gfCNCPoint6[2430] = {X 578.0214, Y 47.7529, Z -8.0000, A 0.000, B 0.000, C 0.000 }
gfCNCPoint6[2431] = {X 577.4979, Y 46.9263, Z -8.0000, A 0.000, B 0.000, C 0.000 }
gfCNCPoint6[2432] = {X 577.4375, Y 46.7968, Z -8.0000, A 0.000, B 0.000, C 0.000 }
gfCNCPoint6[2433] = {X 577.3813, Y 46.6655, Z -8.0000, A 0.000, B 0.000, C 0.000 }
gfCNCPoint6[2434] = {X 572.1002, Y 33.7518, Z -8.0000, A 0.000, B 0.000, C 0.000 }
gfCNCPoint6[2435] = {X 572.1003, Y 35.0200, Z -8.0000, A 0.000, B 0.000, C 0.000 }
gfCNCPoint6[2436] = {X 572.1004, Y 40.7342, Z -8.0000, A 0.000, B 0.000, C 0.000 }
gfCNCPoint6[2437] = {X 572.7444, Y 41.4232, Z -8.0000, A 0.000, B 0.000, C 0.000 }
gfCNCPoint6[2438] = {X 573.2268, Y 42.2337, Z -8.0000, A 0.000, B 0.000, C 0.000 }
gfCNCPoint6[2439] = {X 573.5254, Y 43.1283, Z -8.0000, A 0.000, B 0.000, C 0.000 }
gfCNCPoint6[2440] = {X 573.6264, Y 44.0660, Z -8.0000, A 0.000, B 0.000, C 0.000 }
gfCNCPoint6[2441] = {X 573.6264, Y 45.0000, Z -8.0000, A 0.000, B 0.000, C 0.000 }
gfCNCPoint6[2442] = {X 573.5140, Y 45.9884, Z -8.0000, A 0.000, B 0.000, C 0.000 }
gfCNCPoint6[2443] = {X 573.1824, Y 46.9263, Z -8.0000, A 0.000, B 0.000, C 0.000 }
gfCNCPoint6[2444] = {X 572.6569, Y 47.7553, Z -8.0000, A 0.000, B 0.000, C 0.000 }
gfCNCPoint6[2445] = {X 571.9608, Y 48.4472, Z -8.0000, A 0.000, B 0.000, C 0.000 }
gfCNCPoint6[2446] = {X 571.1286, Y 48.9676, Z -8.0000, A 0.000, B 0.000, C 0.000 }
gfCNCPoint6[2447] = {X 570.2018, Y 49.2905, Z -8.0000, A 0.000, B 0.000, C 0.000 }
gfCNCPoint6[2448] = {X 569.2264, Y 49.4000, Z -8.0000, A 0.000, B 0.000, C 0.000 }
gfCNCPoint6[2449] = {X 562.4443, Y 49.4000, Z -8.0000, A 0.000, B 0.000, C 0.000 }
gfCNCPoint6[2450] = {X 561.4652, Y 49.2897, Z -8.0000, A 0.000, B 0.000, C 0.000 }
gfCNCPoint6[2451] = {X 560.5352, Y 48.9643, Z -8.0000, A 0.000, B 0.000, C 0.000 }
gfCNCPoint6[2452] = {X 559.7009, Y 48.4401, Z -8.0000, A 0.000, B 0.000, C 0.000 }
gfCNCPoint6[2453] = {X 559.0042, Y 47.7434, Z -8.0000, A 0.000, B 0.000, C 0.000 }
gfCNCPoint6[2454] = {X 558.4800, Y 46.9091, Z -8.0000, A 0.000, B 0.000, C 0.000 }
gfCNCPoint6[2455] = {X 558.1546, Y 45.9791, Z -8.0000, A 0.000, B 0.000, C 0.000 }
gfCNCPoint6[2456] = {X 558.0443, Y 45.0000, Z -8.0000, A 0.000, B 0.000, C 0.000 }
gfCNCPoint6[2457] = {X 558.0443, Y 44.0647, Z -8.0000, A 0.000, B 0.000, C 0.000 }
gfCNCPoint6[2458] = {X 558.1476, Y 43.1278, Z -8.0000, A 0.000, B 0.000, C 0.000 }
gfCNCPoint6[2459] = {X 558.4468, Y 42.2339, Z -8.0000, A 0.000, B 0.000, C 0.000 }
gfCNCPoint6[2460] = {X 558.9284, Y 41.4236, Z -8.0000, A 0.000, B 0.000, C 0.000 }
gfCNCPoint6[2461] = {X 559.5706, Y 40.7336, Z -8.0000, A 0.000, B 0.000, C 0.000 }
gfCNCPoint6[2462] = {X 559.5710, Y 9.2664, Z -8.0000, A 0.000, B 0.000, C 0.000 }
gfCNCPoint6[2463] = {X 558.9267, Y 8.5773, Z -8.0000, A 0.000, B 0.000, C 0.000 }
gfCNCPoint6[2464] = {X 558.4441, Y 7.7667, Z -8.0000, A 0.000, B 0.000, C 0.000 }
gfCNCPoint6[2465] = {X 558.1454, Y 6.8719, Z -8.0000, A 0.000, B 0.000, C 0.000 }
gfCNCPoint6[2466] = {X 558.0443, Y 5.9340, Z -8.0000, A 0.000, B 0.000, C 0.000 }
gfCNCPoint6[2467] = {X 558.0443, Y 5.0000, Z -8.0000, A 0.000, B 0.000, C 0.000 }
gfCNCPoint6[2468] = {X 558.1353, Y 4.1096, Z -8.0000, A 0.000, B 0.000, C 0.000 }
gfCNCPoint6[2469] = {X 558.4047, Y 3.2561, Z -8.0000, A 0.000, B 0.000, C 0.000 }
gfCNCPoint6[2470] = {X 558.9156, Y 2.3717, Z -8.0000, A 0.000, B 0.000, C 0.000 }
gfCNCPoint6[2471] = {X 559.6166, Y 1.6289, Z -8.0000, A 0.000, B 0.000, C 0.000 }
gfCNCPoint6[2472] = {X 560.4700, Y 1.0678, Z -8.0000, A 0.000, B 0.000, C 0.000 }
gfCNCPoint6[2473] = {X 561.4298, Y 0.7185, Z -8.0000, A 0.000, B 0.000, C 0.000 }
gfCNCPoint6[2474] = {X 562.4443, Y 0.6000, Z -8.0000, A 0.000, B 0.000, C 0.000 }
gfCNCPoint6[2475] = {X 570.9376, Y 0.6000, Z -8.0000, A 0.000, B 0.000, C 0.000 }
gfCNCPoint6[2476] = {X 571.9520, Y 0.7185, Z -8.0000, A 0.000, B 0.000, C 0.000 }
gfCNCPoint6[2477] = {X 572.9118, Y 1.0678, Z -8.0000, A 0.000, B 0.000, C 0.000 }
gfCNCPoint6[2478] = {X 573.7652, Y 1.6289, Z -8.0000, A 0.000, B 0.000, C 0.000 }
gfCNCPoint6[2479] = {X 574.4663, Y 2.3717, Z -8.0000, A 0.000, B 0.000, C 0.000 }
gfCNCPoint6[2480] = {X 574.9772, Y 3.2561, Z -8.0000, A 0.000, B 0.000, C 0.000 }
gfCNCPoint6[2481] = {X 575.2465, Y 4.1096, Z -8.0000, A 0.000, B 0.000, C 0.000 }
gfCNCPoint6[2482] = {X 575.3376, Y 5.0000, Z -8.0000, A 0.000, B 0.000, C 0.000 }
gfCNCPoint6[2483] = {X 575.3372, Y 5.9910, Z -8.0000, A 0.000, B 0.000, C 0.000 }
gfCNCPoint6[2484] = {X 575.2578, Y 6.7682, Z -8.0000, A 0.000, B 0.000, C 0.000 }
gfCNCPoint6[2485] = {X 575.0421, Y 7.5192, Z -8.0000, A 0.000, B 0.000, C 0.000 }
gfCNCPoint6[2486] = {X 574.6971, Y 8.2201, Z -8.0000, A 0.000, B 0.000, C 0.000 }
gfCNCPoint6[2487] = {X 575.2866, Y 9.6556, Z -8.0000, A 0.000, B 0.000, C 0.000 }
gfCNCPoint6[2488] = {X 578.9730, Y 18.7089, Z -8.0000, A 0.000, B 0.000, C 0.000 }
gfCNCPoint6[2489] = {X 580.9325, Y 23.5210, Z -8.0000, A 0.000, B 0.000, C 0.000 }
gfCNCPoint6[2490] = {X 581.1912, Y 24.1565, Z -8.0000, A 0.000, B 0.000, C 0.000 }
gfCNCPoint6[2491] = {X 581.4509, Y 23.5214, Z -8.0000, A 0.000, B 0.000, C 0.000 }
gfCNCPoint6[2492] = {X 587.7566, Y 8.0994, Z -8.0000, A 0.000, B 0.000, C 0.000 }
gfCNCPoint6[2493] = {X 587.4433, Y 7.4139, Z -8.0000, A 0.000, B 0.000, C 0.000 }
gfCNCPoint6[2494] = {X 587.2515, Y 6.6850, Z -8.0000, A 0.000, B 0.000, C 0.000 }
gfCNCPoint6[2495] = {X 587.1870, Y 5.9340, Z -8.0000, A 0.000, B 0.000, C 0.000 }
gfCNCPoint6[2496] = {X 587.1870, Y 5.0000, Z -8.0000, A 0.000, B 0.000, C 0.000 }
gfCNCPoint6[2497] = {X 587.2780, Y 4.1096, Z -8.0000, A 0.000, B 0.000, C 0.000 }
gfCNCPoint6[2498] = {X 587.5473, Y 3.2561, Z -8.0000, A 0.000, B 0.000, C 0.000 }
gfCNCPoint6[2499] = {X 588.0582, Y 2.3717, Z -8.0000, A 0.000, B 0.000, C 0.000 }
gfCNCPoint6[2500] = {X 588.7593, Y 1.6289, Z -8.0000, A 0.000, B 0.000, C 0.000 }
gfCNCPoint6[2501] = {X 589.6127, Y 1.0678, Z -8.0000, A 0.000, B 0.000, C 0.000 }
gfCNCPoint6[2502] = {X 590.5725, Y 0.7185, Z -8.0000, A 0.000, B 0.000, C 0.000 }
gfCNCPoint6[2503] = {X 591.5870, Y 0.6000, Z -8.0000, A 0.000, B 0.000, C 0.000 }
gfCNCPoint6[2504] = {X 600.0000, Y 0.6000, Z -8.0000, A 0.000, B 0.000, C 0.000 }
gfCNCPoint6[2505] = {X 600.8721, Y 0.6873, Z -8.0000, A 0.000, B 0.000, C 0.000 }
gfCNCPoint6[2506] = {X 601.7095, Y 0.9457, Z -8.0000, A 0.000, B 0.000, C 0.000 }
gfCNCPoint6[2507] = {X 602.4791, Y 1.3649, Z -8.0000, A 0.000, B 0.000, C 0.000 }
gfCNCPoint6[2508] = {X 603.1504, Y 1.9284, Z -8.0000, A 0.000, B 0.000, C 0.000 }
gfCNCPoint6[2509] = {X 603.6967, Y 2.6137, Z -8.0000, A 0.000, B 0.000, C 0.000 }
gfCNCPoint6[2510] = {X 603.6967, Y 1.8143, Z -8.0000, A 0.000, B 0.000, C 0.000 }
gfCNCPoint6[2511] = {X 602.9514, Y 1.1137, Z -8.0000, A 0.000, B 0.000, C 0.000 }
gfCNCPoint6[2512] = {X 602.0764, Y 0.5838, Z -8.0000, A 0.000, B 0.000, C 0.000 }
gfCNCPoint6[2513] = {X 601.1102, Y 0.2480, Z -8.0000, A 0.000, B 0.000, C 0.000 }
gfCNCPoint6[2514] = {X 600.0953, Y 0.1209, Z -8.0000, A 0.000, B 0.000, C 0.000 }
gfCNCPoint6[2515] = {X 600.0950, Y -0.0186, Z -8.0000, A 0.000, B 0.000, C 0.000 }
gfCNCPoint6[2516] = {X 600.0672, Y -0.0699, Z -8.0000, A 0.000, B 0.000, C 0.000 }
gfCNCPoint6[2517] = {X 600.0147, Y -0.0952, Z -8.0000, A 0.000, B 0.000, C 0.000 }
gfCNCPoint6[2518] = {X 580.1328, Y -0.0952, Z -8.0000, A 0.000, B 0.000, C 0.000 }
gfCNCPoint6[2519] = {X 580.1328, Y 4.7048, Z -8.0000, A 0.000, B 0.000, C 0.000 }
gfCNCPoint6[2520] = {X 580.1364, Y 4.8524, Z -8.0000, A 0.000, B 0.000, C 0.000 }
gfCNCPoint6[2521] = {X 580.1376, Y 5.0000, Z -8.0000, A 0.000, B 0.000, C 0.000 }
gfCNCPoint6[2522] = {X 580.1376, Y 5.9339, Z -8.0000, A 0.000, B 0.000, C 0.000 }
gfCNCPoint6[2523] = {X 580.0686, Y 7.0584, Z -8.0000, A 0.000, B 0.000, C 0.000 }
gfCNCPoint6[2524] = {X 579.8627, Y 8.1660, Z -8.0000, A 0.000, B 0.000, C 0.000 }
gfCNCPoint6[2525] = {X 581.2004, Y 11.4512, Z -8.0000, A 0.000, B 0.000, C 0.000 }
gfCNCPoint6[2526] = {X 582.6182, Y 7.9837, Z -8.0000, A 0.000, B 0.000, C 0.000 }
gfCNCPoint6[2527] = {X 582.4488, Y 6.9991, Z -8.0000, A 0.000, B 0.000, C 0.000 }
gfCNCPoint6[2528] = {X 582.3872, Y 6.0018, Z -8.0000, A 0.000, B 0.000, C 0.000 }
gfCNCPoint6[2529] = {X 582.3870, Y 5.0000, Z -8.0000, A 0.000, B 0.000, C 0.000 }
gfCNCPoint6[2530] = {X 582.3881, Y 4.8524, Z -8.0000, A 0.000, B 0.000, C 0.000 }
gfCNCPoint6[2531] = {X 582.3917, Y 4.7048, Z -8.0000, A 0.000, B 0.000, C 0.000 }
gfCNCPoint6[2532] = {X 580.1328, Y 4.7048, Z -8.0000, A 0.000, B 0.000, C 0.000 }
gfCNCPoint6[2533] = {X 580.1328, Y 2.3048, Z -8.0000, A 0.000, B 0.000, C 0.000 }
gfCNCPoint6[2534] = {X 577.1806, Y 2.3048, Z -8.0000, A 0.000, B 0.000, C 0.000 }
gfCNCPoint6[2535] = {X 577.5739, Y 3.5173, Z -8.0000, A 0.000, B 0.000, C 0.000 }
gfCNCPoint6[2536] = {X 577.7341, Y 4.7818, Z -8.0000, A 0.000, B 0.000, C 0.000 }
gfCNCPoint6[2537] = {X 577.7367, Y 4.8909, Z -8.0000, A 0.000, B 0.000, C 0.000 }
gfCNCPoint6[2538] = {X 577.7376, Y 5.0000, Z -8.0000, A 0.000, B 0.000, C 0.000 }
gfCNCPoint6[2539] = {X 577.7376, Y 5.9339, Z -8.0000, A 0.000, B 0.000, C 0.000 }
gfCNCPoint6[2540] = {X 577.6319, Y 7.1280, Z -8.0000, A 0.000, B 0.000, C 0.000 }
gfCNCPoint6[2541] = {X 577.3182, Y 8.2850, Z -8.0000, A 0.000, B 0.000, C 0.000 }
gfCNCPoint6[2542] = {X 577.5061, Y 8.7426, Z -8.0000, A 0.000, B 0.000, C 0.000 }
gfCNCPoint6[2543] = {X 581.1958, Y 17.8038, Z -8.0000, A 0.000, B 0.000, C 0.000 }
gfCNCPoint6[2544] = {X 585.1513, Y 8.1300, Z -8.0000, A 0.000, B 0.000, C 0.000 }
gfCNCPoint6[2545] = {X 584.8834, Y 7.0753, Z -8.0000, A 0.000, B 0.000, C 0.000 }
gfCNCPoint6[2546] = {X 584.7872, Y 5.9914, Z -8.0000, A 0.000, B 0.000, C 0.000 }
gfCNCPoint6[2547] = {X 584.7870, Y 5.0000, Z -8.0000, A 0.000, B 0.000, C 0.000 }
gfCNCPoint6[2548] = {X 584.7878, Y 4.8909, Z -8.0000, A 0.000, B 0.000, C 0.000 }
gfCNCPoint6[2549] = {X 584.7905, Y 4.7818, Z -8.0000, A 0.000, B 0.000, C 0.000 }
gfCNCPoint6[2550] = {X 584.9506, Y 3.5173, Z -8.0000, A 0.000, B 0.000, C 0.000 }
gfCNCPoint6[2551] = {X 585.3439, Y 2.3048, Z -8.0000, A 0.000, B 0.000, C 0.000 }
gfCNCPoint6[2552] = {X 580.1328, Y 2.3048, Z -8.0000, A 0.000, B 0.000, C 0.000 }
gfCNCPoint6[2553] = {X 580.1328, Y -0.0952, Z -8.0000, A 0.000, B 0.000, C 0.000 }
gfCNCPoint6[2554] = {X 351.5709, Y -0.0952, Z -8.0000, A 0.000, B 0.000, C 0.000 }
gfCNCPoint6[2555] = {X 351.4056, Y -0.1263, Z -8.0000, A 0.000, B 0.000, C 0.000 }
gfCNCPoint6[2556] = {X 348.9077, Y -0.4729, Z -8.0000, A 0.000, B 0.000, C 0.000 }
gfCNCPoint6[2557] = {X 346.3883, Y -0.5836, Z -8.0000, A 0.000, B 0.000, C 0.000 }
gfCNCPoint6[2558] = {X 343.8697, Y -0.4573, Z -8.0000, A 0.000, B 0.000, C 0.000 }
gfCNCPoint6[2559] = {X 341.3740, Y -0.0952, Z -8.0000, A 0.000, B 0.000, C 0.000 }
gfCNCPoint6[2560] = {X -0.0147, Y -0.0952, Z -8.0000, A 0.000, B 0.000, C 0.000 }
gfCNCPoint6[2561] = {X -0.0672, Y -0.0699, Z -8.0000, A 0.000, B 0.000, C 0.000 }
gfCNCPoint6[2562] = {X -0.0950, Y -0.0186, Z -8.0000, A 0.000, B 0.000, C 0.000 }
gfCNCPoint6[2563] = {X -0.0967, Y 0.8568, Z -8.0000, A 0.000, B 0.000, C 0.000 }
gfCNCPoint6[2564] = {X -0.0967, Y 8.7891, Z -8.0000, A 0.000, B 0.000, C 0.000 }
gfCNCPoint6[2565] = {X -0.7634, Y 8.9979, Z -8.0000, A 0.000, B 0.000, C 0.000 }
gfCNCPoint6[2566] = {X -1.3934, Y 9.2998, Z -8.0000, A 0.000, B 0.000, C 0.000 }
gfCNCPoint6[2567] = {X -1.9904, Y 9.6404, Z -8.0000, A 0.000, B 0.000, C 0.000 }
gfCNCPoint6[2568] = {X -2.6455, Y 10.0885, Z -8.0000, A 0.000, B 0.000, C 0.000 }
gfCNCPoint6[2569] = {X -3.2194, Y 10.6368, Z -8.0000, A 0.000, B 0.000, C 0.000 }
gfCNCPoint6[2570] = {X -3.6967, Y 11.2708, Z -8.0000, A 0.000, B 0.000, C 0.000 }
gfCNCPoint6[2571] = {X -3.6967, Y 12.3466, Z -8.0000, A 0.000, B 0.000, C 0.000 }
gfCNCPoint6[2572] = {X -3.2334, Y 11.4386, Z -8.0000, A 0.000, B 0.000, C 0.000 }
gfCNCPoint6[2573] = {X -2.5735, Y 10.6616, Z -8.0000, A 0.000, B 0.000, C 0.000 }
gfCNCPoint6[2574] = {X -1.7526, Y 10.0573, Z -8.0000, A 0.000, B 0.000, C 0.000 }
gfCNCPoint6[2575] = {X -1.0994, Y 9.6852, Z -8.0000, A 0.000, B 0.000, C 0.000 }
gfCNCPoint6[2576] = {X -0.1608, Y 9.3012, Z -8.0000, A 0.000, B 0.000, C 0.000 }
gfCNCPoint6[2577] = {X 0.8408, Y 9.1423, Z -8.0000, A 0.000, B 0.000, C 0.000 }
gfCNCPoint6[2578] = {X 1.8521, Y 9.2169, Z -8.0000, A 0.000, B 0.000, C 0.000 }
gfCNCPoint6[2579] = {X 2.2301, Y 9.3067, Z -8.0000, A 0.000, B 0.000, C 0.000 }
gfCNCPoint6[2580] = {X 2.5987, Y 9.4295, Z -8.0000, A 0.000, B 0.000, C 0.000 }
gfCNCPoint6[2581] = {X 3.4585, Y 9.0449, Z -8.0000, A 0.000, B 0.000, C 0.000 }
gfCNCPoint6[2582] = {X 5.5423, Y 8.2600, Z -8.0000, A 0.000, B 0.000, C 0.000 }
gfCNCPoint6[2583] = {X 7.6901, Y 7.6725, Z -8.0000, A 0.000, B 0.000, C 0.000 }
gfCNCPoint6[2584] = {X 9.8833, Y 7.2876, Z -8.0000, A 0.000, B 0.000, C 0.000 }
gfCNCPoint6[2585] = {X 12.1029, Y 7.1087, Z -8.0000, A 0.000, B 0.000, C 0.000 }
gfCNCPoint6[2586] = {X 14.3294, Y 7.1373, Z -8.0000, A 0.000, B 0.000, C 0.000 }
gfCNCPoint6[2587] = {X 16.5436, Y 7.3732, Z -8.0000, A 0.000, B 0.000, C 0.000 }
gfCNCPoint6[2588] = {X 18.2874, Y 7.7294, Z -8.0000, A 0.000, B 0.000, C 0.000 }
gfCNCPoint6[2589] = {X 19.9860, Y 8.2610, Z -8.0000, A 0.000, B 0.000, C 0.000 }
gfCNCPoint6[2590] = {X 21.6217, Y 8.9626, Z -8.0000, A 0.000, B 0.000, C 0.000 }
gfCNCPoint6[2591] = {X 23.1776, Y 9.8268, Z -8.0000, A 0.000, B 0.000, C 0.000 }
gfCNCPoint6[2592] = {X 24.6376, Y 10.8447, Z -8.0000, A 0.000, B 0.000, C 0.000 }
gfCNCPoint6[2593] = {X 25.7303, Y 11.8004, Z -8.0000, A 0.000, B 0.000, C 0.000 }
gfCNCPoint6[2594] = {X 26.7104, Y 12.8713, Z -8.0000, A 0.000, B 0.000, C 0.000 }
gfCNCPoint6[2595] = {X 27.5658, Y 14.0441, Z -8.0000, A 0.000, B 0.000, C 0.000 }
gfCNCPoint6[2596] = {X 28.2861, Y 15.3044, Z -8.0000, A 0.000, B 0.000, C 0.000 }
gfCNCPoint6[2597] = {X 28.8624, Y 16.6368, Z -8.0000, A 0.000, B 0.000, C 0.000 }
gfCNCPoint6[2598] = {X 29.3390, Y 18.3013, Z -8.0000, A 0.000, B 0.000, C 0.000 }
gfCNCPoint6[2599] = {X 29.6217, Y 20.0095, Z -8.0000, A 0.000, B 0.000, C 0.000 }
gfCNCPoint6[2600] = {X 29.7069, Y 21.7388, Z -8.0000, A 0.000, B 0.000, C 0.000 }
gfCNCPoint6[2601] = {X 29.5934, Y 23.4664, Z -8.0000, A 0.000, B 0.000, C 0.000 }
gfCNCPoint6[2602] = {X 29.2828, Y 25.1698, Z -8.0000, A 0.000, B 0.000, C 0.000 }
gfCNCPoint6[2603] = {X 28.7910, Y 26.7456, Z -8.0000, A 0.000, B 0.000, C 0.000 }
gfCNCPoint6[2604] = {X 28.0838, Y 28.2372, Z -8.0000, A 0.000, B 0.000, C 0.000 }
gfCNCPoint6[2605] = {X 27.1749, Y 29.6152, Z -8.0000, A 0.000, B 0.000, C 0.000 }
gfCNCPoint6[2606] = {X 26.3579, Y 30.5723, Z -8.0000, A 0.000, B 0.000, C 0.000 }
gfCNCPoint6[2607] = {X 25.4435, Y 31.4368, Z -8.0000, A 0.000, B 0.000, C 0.000 }
gfCNCPoint6[2608] = {X 25.6940, Y 31.5324, Z -8.0000, A 0.000, B 0.000, C 0.000 }
gfCNCPoint6[2609] = {X 25.9383, Y 31.6432, Z -8.0000, A 0.000, B 0.000, C 0.000 }
gfCNCPoint6[2610] = {X 26.6629, Y 32.0904, Z -8.0000, A 0.000, B 0.000, C 0.000 }
gfCNCPoint6[2611] = {X 27.2878, Y 32.6689, Z -8.0000, A 0.000, B 0.000, C 0.000 }
gfCNCPoint6[2612] = {X 27.6592, Y 33.1494, Z -8.0000, A 0.000, B 0.000, C 0.000 }
gfCNCPoint6[2613] = {X 27.9608, Y 33.6765, Z -8.0000, A 0.000, B 0.000, C 0.000 }
gfCNCPoint6[2614] = {X 30.9820, Y 39.9182, Z -8.0000, A 0.000, B 0.000, C 0.000 }
gfCNCPoint6[2615] = {X 31.3085, Y 40.8441, Z -8.0000, A 0.000, B 0.000, C 0.000 }
gfCNCPoint6[2616] = {X 31.4215, Y 41.8194, Z -8.0000, A 0.000, B 0.000, C 0.000 }
gfCNCPoint6[2617] = {X 31.3155, Y 42.7955, Z -8.0000, A 0.000, B 0.000, C 0.000 }
gfCNCPoint6[2618] = {X 30.9956, Y 43.7238, Z -8.0000, A 0.000, B 0.000, C 0.000 }
gfCNCPoint6[2619] = {X 30.4779, Y 44.5580, Z -8.0000, A 0.000, B 0.000, C 0.000 }
gfCNCPoint6[2620] = {X 29.7880, Y 45.2567, Z -8.0000, A 0.000, B 0.000, C 0.000 }
gfCNCPoint6[2621] = {X 29.2521, Y 45.6900, Z -8.0000, A 0.000, B 0.000, C 0.000 }
gfCNCPoint6[2622] = {X 28.5416, Y 46.1592, Z -8.0000, A 0.000, B 0.000, C 0.000 }
gfCNCPoint6[2623] = {X 27.7541, Y 46.4832, Z -8.0000, A 0.000, B 0.000, C 0.000 }
gfCNCPoint6[2624] = {X 26.9190, Y 46.6497, Z -8.0000, A 0.000, B 0.000, C 0.000 }
gfCNCPoint6[2625] = {X 26.0675, Y 46.6526, Z -8.0000, A 0.000, B 0.000, C 0.000 }
gfCNCPoint6[2626] = {X 25.2313, Y 46.4918, Z -8.0000, A 0.000, B 0.000, C 0.000 }
gfCNCPoint6[2627] = {X 23.4347, Y 47.4365, Z -8.0000, A 0.000, B 0.000, C 0.000 }
gfCNCPoint6[2628] = {X 21.5774, Y 48.2554, Z -8.0000, A 0.000, B 0.000, C 0.000 }
gfCNCPoint6[2629] = {X 19.6682, Y 48.9447, Z -8.0000, A 0.000, B 0.000, C 0.000 }
gfCNCPoint6[2630] = {X 17.7217, Y 49.4942, Z -8.0000, A 0.000, B 0.000, C 0.000 }
gfCNCPoint6[2631] = {X 15.7341, Y 49.8692, Z -8.0000, A 0.000, B 0.000, C 0.000 }
gfCNCPoint6[2632] = {X 13.7212, Y 50.0669, Z -8.0000, A 0.000, B 0.000, C 0.000 }
gfCNCPoint6[2633] = {X 11.6986, Y 50.0856, Z -8.0000, A 0.000, B 0.000, C 0.000 }
gfCNCPoint6[2634] = {X 9.6824, Y 49.9253, Z -8.0000, A 0.000, B 0.000, C 0.000 }
gfCNCPoint6[2635] = {X 7.6882, Y 49.5872, Z -8.0000, A 0.000, B 0.000, C 0.000 }
gfCNCPoint6[2636] = {X 6.2182, Y 49.2062, Z -8.0000, A 0.000, B 0.000, C 0.000 }
gfCNCPoint6[2637] = {X 4.7886, Y 48.6940, Z -8.0000, A 0.000, B 0.000, C 0.000 }
gfCNCPoint6[2638] = {X 3.4111, Y 48.0546, Z -8.0000, A 0.000, B 0.000, C 0.000 }
gfCNCPoint6[2639] = {X 1.9573, Y 47.2030, Z -8.0000, A 0.000, B 0.000, C 0.000 }
gfCNCPoint6[2640] = {X 0.5963, Y 46.2099, Z -8.0000, A 0.000, B 0.000, C 0.000 }
gfCNCPoint6[2641] = {X -0.5425, Y 45.1859, Z -8.0000, A 0.000, B 0.000, C 0.000 }
gfCNCPoint6[2642] = {X -1.5540, Y 44.0360, Z -8.0000, A 0.000, B 0.000, C 0.000 }
gfCNCPoint6[2643] = {X -2.4244, Y 42.7759, Z -8.0000, A 0.000, B 0.000, C 0.000 }
gfCNCPoint6[2644] = {X -3.1419, Y 41.4230, Z -8.0000, A 0.000, B 0.000, C 0.000 }
gfCNCPoint6[2645] = {X -3.6967, Y 39.9955, Z -8.0000, A 0.000, B 0.000, C 0.000 }
gfCNCPoint6[2646] = {X -3.6967, Y 41.3567, Z -8.0000, A 0.000, B 0.000, C 0.000 }
gfCNCPoint6[2647] = {X -3.0106, Y 42.7271, Z -8.0000, A 0.000, B 0.000, C 0.000 }
gfCNCPoint6[2648] = {X -2.1745, Y 44.0116, Z -8.0000, A 0.000, B 0.000, C 0.000 }
gfCNCPoint6[2649] = {X -1.1991, Y 45.1937, Z -8.0000, A 0.000, B 0.000, C 0.000 }
gfCNCPoint6[2650] = {X -0.0967, Y 46.2584, Z -8.0000, A 0.000, B 0.000, C 0.000 }
gfCNCPoint6[2651] = {X -0.0967, Y 99.1432, Z -8.0000, A 0.000, B 0.000, C 0.000 }
gfCNCPoint6[2652] = {X -0.0950, Y 100.0186, Z -8.0000, A 0.000, B 0.000, C 0.000 }
gfCNCPoint6[2653] = {X -0.0672, Y 100.0699, Z -8.0000, A 0.000, B 0.000, C 0.000 }
gfCNCPoint6[2654] = {X -0.0147, Y 100.0952, Z -8.0000, A 0.000, B 0.000, C 0.000 }
gfCNCPoint6[2655] = {X 120.5927, Y 100.0952, Z -8.0000, A 0.000, B 0.000, C 0.000 }
gfCNCPoint6[2656] = {X 121.0614, Y 100.8813, Z -8.0000, A 0.000, B 0.000, C 0.000 }
gfCNCPoint6[2657] = {X 121.6688, Y 101.5661, Z -8.0000, A 0.000, B 0.000, C 0.000 }
gfCNCPoint6[2658] = {X 122.3933, Y 102.1255, Z -8.0000, A 0.000, B 0.000, C 0.000 }
gfCNCPoint6[2659] = {X 123.2095, Y 102.5397, Z -8.0000, A 0.000, B 0.000, C 0.000 }
gfCNCPoint6[2660] = {X 124.0887, Y 102.7942, Z -8.0000, A 0.000, B 0.000, C 0.000 }
gfCNCPoint6[2661] = {X 125.0000, Y 102.8800, Z -8.0000, A 0.000, B 0.000, C 0.000 }
gfCNCPoint6[2662] = {X 143.7791, Y 102.8800, Z -8.0000, A 0.000, B 0.000, C 0.000 }
gfCNCPoint6[2663] = {X 144.6904, Y 102.7942, Z -8.0000, A 0.000, B 0.000, C 0.000 }
gfCNCPoint6[2664] = {X 145.5696, Y 102.5397, Z -8.0000, A 0.000, B 0.000, C 0.000 }
gfCNCPoint6[2665] = {X 146.3858, Y 102.1255, Z -8.0000, A 0.000, B 0.000, C 0.000 }
gfCNCPoint6[2666] = {X 147.1104, Y 101.5661, Z -8.0000, A 0.000, B 0.000, C 0.000 }
gfCNCPoint6[2667] = {X 147.7177, Y 100.8813, Z -8.0000, A 0.000, B 0.000, C 0.000 }
gfCNCPoint6[2668] = {X 148.1865, Y 100.0952, Z -8.0000, A 0.000, B 0.000, C 0.000 }
gfCNCPoint6[2669] = {X 150.8390, Y 100.0952, Z -8.0000, A 0.000, B 0.000, C 0.000 }
gfCNCPoint6[2670] = {X 150.8390, Y 95.2952, Z -8.0000, A 0.000, B 0.000, C 0.000 }
gfCNCPoint6[2671] = {X 187.9256, Y 95.2952, Z -8.0000, A 0.000, B 0.000, C 0.000 }
gfCNCPoint6[2672] = {X 187.9777, Y 95.0991, Z -8.0000, A 0.000, B 0.000, C 0.000 }
gfCNCPoint6[2673] = {X 188.0352, Y 94.9045, Z -8.0000, A 0.000, B 0.000, C 0.000 }
gfCNCPoint6[2674] = {X 187.2619, Y 94.0602, Z -8.0000, A 0.000, B 0.000, C 0.000 }
gfCNCPoint6[2675] = {X 151.4055, Y 94.0602, Z -8.0000, A 0.000, B 0.000, C 0.000 }
gfCNCPoint6[2676] = {X 150.7069, Y 94.8343, Z -8.0000, A 0.000, B 0.000, C 0.000 }
gfCNCPoint6[2677] = {X 150.7767, Y 95.0636, Z -8.0000, A 0.000, B 0.000, C 0.000 }
gfCNCPoint6[2678] = {X 150.8390, Y 95.2952, Z -8.0000, A 0.000, B 0.000, C 0.000 }
gfCNCPoint6[2679] = {X 150.8390, Y 97.6952, Z -8.0000, A 0.000, B 0.000, C 0.000 }
gfCNCPoint6[2680] = {X 190.1070, Y 97.6952, Z -8.0000, A 0.000, B 0.000, C 0.000 }
gfCNCPoint6[2681] = {X 190.1070, Y 97.0659, Z -8.0000, A 0.000, B 0.000, C 0.000 }
gfCNCPoint6[2682] = {X 190.1938, Y 96.1495, Z -8.0000, A 0.000, B 0.000, C 0.000 }
gfCNCPoint6[2683] = {X 190.4511, Y 95.2657, Z -8.0000, A 0.000, B 0.000, C 0.000 }
gfCNCPoint6[2684] = {X 190.8699, Y 94.4460, Z -8.0000, A 0.000, B 0.000, C 0.000 }
gfCNCPoint6[2685] = {X 188.3182, Y 91.6602, Z -8.0000, A 0.000, B 0.000, C 0.000 }
gfCNCPoint6[2686] = {X 150.3387, Y 91.6602, Z -8.0000, A 0.000, B 0.000, C 0.000 }
gfCNCPoint6[2687] = {X 147.8648, Y 94.4010, Z -8.0000, A 0.000, B 0.000, C 0.000 }
gfCNCPoint6[2688] = {X 148.2994, Y 95.2322, Z -8.0000, A 0.000, B 0.000, C 0.000 }
gfCNCPoint6[2689] = {X 148.5675, Y 96.1310, Z -8.0000, A 0.000, B 0.000, C 0.000 }
gfCNCPoint6[2690] = {X 148.6591, Y 97.0644, Z -8.0000, A 0.000, B 0.000, C 0.000 }
gfCNCPoint6[2691] = {X 148.6591, Y 97.6952, Z -8.0000, A 0.000, B 0.000, C 0.000 }
gfCNCPoint6[2692] = {X 150.8390, Y 97.6952, Z -8.0000, A 0.000, B 0.000, C 0.000 }
gfCNCPoint6[2693] = {X 150.8390, Y 100.0952, Z -8.0000, A 0.000, B 0.000, C 0.000 }
gfCNCPoint6[2694] = {X 190.5796, Y 100.0952, Z -8.0000, A 0.000, B 0.000, C 0.000 }
gfCNCPoint6[2695] = {X 191.0484, Y 100.8813, Z -8.0000, A 0.000, B 0.000, C 0.000 }
gfCNCPoint6[2696] = {X 191.6557, Y 101.5661, Z -8.0000, A 0.000, B 0.000, C 0.000 }
gfCNCPoint6[2697] = {X 192.3802, Y 102.1255, Z -8.0000, A 0.000, B 0.000, C 0.000 }
gfCNCPoint6[2698] = {X 193.1965, Y 102.5397, Z -8.0000, A 0.000, B 0.000, C 0.000 }
gfCNCPoint6[2699] = {X 194.0757, Y 102.7942, Z -8.0000, A 0.000, B 0.000, C 0.000 }
gfCNCPoint6[2700] = {X 194.9870, Y 102.8800, Z -8.0000, A 0.000, B 0.000, C 0.000 }
gfCNCPoint6[2701] = {X 212.6141, Y 102.8800, Z -8.0000, A 0.000, B 0.000, C 0.000 }
gfCNCPoint6[2702] = {X 213.0066, Y 102.8642, Z -8.0000, A 0.000, B 0.000, C 0.000 }
gfCNCPoint6[2703] = {X 213.3966, Y 102.8169, Z -8.0000, A 0.000, B 0.000, C 0.000 }
gfCNCPoint6[2704] = {X 213.7865, Y 102.8642, Z -8.0000, A 0.000, B 0.000, C 0.000 }
gfCNCPoint6[2705] = {X 214.1790, Y 102.8800, Z -8.0000, A 0.000, B 0.000, C 0.000 }
gfCNCPoint6[2706] = {X 233.4798, Y 102.8800, Z -8.0000, A 0.000, B 0.000, C 0.000 }
gfCNCPoint6[2707] = {X 234.3911, Y 102.7942, Z -8.0000, A 0.000, B 0.000, C 0.000 }
gfCNCPoint6[2708] = {X 235.2703, Y 102.5397, Z -8.0000, A 0.000, B 0.000, C 0.000 }
gfCNCPoint6[2709] = {X 236.0865, Y 102.1255, Z -8.0000, A 0.000, B 0.000, C 0.000 }
gfCNCPoint6[2710] = {X 236.8110, Y 101.5661, Z -8.0000, A 0.000, B 0.000, C 0.000 }
gfCNCPoint6[2711] = {X 237.4184, Y 100.8813, Z -8.0000, A 0.000, B 0.000, C 0.000 }
gfCNCPoint6[2712] = {X 237.8871, Y 100.0952, Z -8.0000, A 0.000, B 0.000, C 0.000 }
gfCNCPoint6[2713] = {X 261.4882, Y 100.0952, Z -8.0000, A 0.000, B 0.000, C 0.000 }
gfCNCPoint6[2714] = {X 261.4882, Y 90.4952, Z -8.0000, A 0.000, B 0.000, C 0.000 }
gfCNCPoint6[2715] = {X 266.0961, Y 90.4952, Z -8.0000, A 0.000, B 0.000, C 0.000 }
gfCNCPoint6[2716] = {X 266.1751, Y 90.3748, Z -8.0000, A 0.000, B 0.000, C 0.000 }
gfCNCPoint6[2717] = {X 266.2556, Y 90.2554, Z -8.0000, A 0.000, B 0.000, C 0.000 }
gfCNCPoint6[2718] = {X 263.5169, Y 89.1818, Z -8.0000, A 0.000, B 0.000, C 0.000 }
gfCNCPoint6[2719] = {X 261.4882, Y 90.4952, Z -8.0000, A 0.000, B 0.000, C 0.000 }
gfCNCPoint6[2720] = {X 261.4882, Y 92.8952, Z -8.0000, A 0.000, B 0.000, C 0.000 }
gfCNCPoint6[2721] = {X 267.4973, Y 92.8952, Z -8.0000, A 0.000, B 0.000, C 0.000 }
gfCNCPoint6[2722] = {X 267.8429, Y 92.2376, Z -8.0000, A 0.000, B 0.000, C 0.000 }
gfCNCPoint6[2723] = {X 268.2378, Y 91.6085, Z -8.0000, A 0.000, B 0.000, C 0.000 }
gfCNCPoint6[2724] = {X 269.1700, Y 90.4463, Z -8.0000, A 0.000, B 0.000, C 0.000 }
gfCNCPoint6[2725] = {X 270.2694, Y 89.4409, Z -8.0000, A 0.000, B 0.000, C 0.000 }
gfCNCPoint6[2726] = {X 270.2694, Y 89.2510, Z -8.0000, A 0.000, B 0.000, C 0.000 }
gfCNCPoint6[2727] = {X 263.2463, Y 86.4979, Z -8.0000, A 0.000, B 0.000, C 0.000 }
gfCNCPoint6[2728] = {X 253.3650, Y 92.8952, Z -8.0000, A 0.000, B 0.000, C 0.000 }
gfCNCPoint6[2729] = {X 261.4882, Y 92.8952, Z -8.0000, A 0.000, B 0.000, C 0.000 }
gfCNCPoint6[2730] = {X 261.4882, Y 95.2952, Z -8.0000, A 0.000, B 0.000, C 0.000 }
gfCNCPoint6[2731] = {X 269.1713, Y 95.2952, Z -8.0000, A 0.000, B 0.000, C 0.000 }
gfCNCPoint6[2732] = {X 269.5515, Y 94.1746, Z -8.0000, A 0.000, B 0.000, C 0.000 }
gfCNCPoint6[2733] = {X 270.1082, Y 93.1304, Z -8.0000, A 0.000, B 0.000, C 0.000 }
gfCNCPoint6[2734] = {X 270.8267, Y 92.1902, Z -8.0000, A 0.000, B 0.000, C 0.000 }
gfCNCPoint6[2735] = {X 271.6880, Y 91.3788, Z -8.0000, A 0.000, B 0.000, C 0.000 }
gfCNCPoint6[2736] = {X 272.6694, Y 90.7176, Z -8.0000, A 0.000, B 0.000, C 0.000 }
gfCNCPoint6[2737] = {X 272.6694, Y 87.6139, Z -8.0000, A 0.000, B 0.000, C 0.000 }
gfCNCPoint6[2738] = {X 262.9757, Y 83.8140, Z -8.0000, A 0.000, B 0.000, C 0.000 }
gfCNCPoint6[2739] = {X 245.2418, Y 95.2952, Z -8.0000, A 0.000, B 0.000, C 0.000 }
gfCNCPoint6[2740] = {X 261.4882, Y 95.2952, Z -8.0000, A 0.000, B 0.000, C 0.000 }
gfCNCPoint6[2741] = {X 261.4882, Y 97.6952, Z -8.0000, A 0.000, B 0.000, C 0.000 }
gfCNCPoint6[2742] = {X 271.3527, Y 97.6952, Z -8.0000, A 0.000, B 0.000, C 0.000 }
gfCNCPoint6[2743] = {X 271.3529, Y 97.0186, Z -8.0000, A 0.000, B 0.000, C 0.000 }
gfCNCPoint6[2744] = {X 271.4810, Y 95.9545, Z -8.0000, A 0.000, B 0.000, C 0.000 }
gfCNCPoint6[2745] = {X 271.8382, Y 94.9440, Z -8.0000, A 0.000, B 0.000, C 0.000 }
gfCNCPoint6[2746] = {X 272.4074, Y 94.0359, Z -8.0000, A 0.000, B 0.000, C 0.000 }
gfCNCPoint6[2747] = {X 273.1610, Y 93.2739, Z -8.0000, A 0.000, B 0.000, C 0.000 }
gfCNCPoint6[2748] = {X 274.0629, Y 92.6949, Z -8.0000, A 0.000, B 0.000, C 0.000 }
gfCNCPoint6[2749] = {X 275.0694, Y 92.3266, Z -8.0000, A 0.000, B 0.000, C 0.000 }
gfCNCPoint6[2750] = {X 275.0694, Y 85.9769, Z -8.0000, A 0.000, B 0.000, C 0.000 }
gfCNCPoint6[2751] = {X 262.7051, Y 81.1301, Z -8.0000, A 0.000, B 0.000, C 0.000 }
gfCNCPoint6[2752] = {X 238.3590, Y 96.8921, Z -8.0000, A 0.000, B 0.000, C 0.000 }
gfCNCPoint6[2753] = {X 238.3598, Y 97.6952, Z -8.0000, A 0.000, B 0.000, C 0.000 }
gfCNCPoint6[2754] = {X 261.4882, Y 97.6952, Z -8.0000, A 0.000, B 0.000, C 0.000 }
gfCNCPoint6[2755] = {X 261.4882, Y 100.0952, Z -8.0000, A 0.000, B 0.000, C 0.000 }
gfCNCPoint6[2756] = {X 271.8253, Y 100.0952, Z -8.0000, A 0.000, B 0.000, C 0.000 }
gfCNCPoint6[2757] = {X 272.2941, Y 100.8813, Z -8.0000, A 0.000, B 0.000, C 0.000 }
gfCNCPoint6[2758] = {X 272.9014, Y 101.5661, Z -8.0000, A 0.000, B 0.000, C 0.000 }
gfCNCPoint6[2759] = {X 273.6260, Y 102.1255, Z -8.0000, A 0.000, B 0.000, C 0.000 }
gfCNCPoint6[2760] = {X 274.4422, Y 102.5397, Z -8.0000, A 0.000, B 0.000, C 0.000 }
gfCNCPoint6[2761] = {X 275.3214, Y 102.7942, Z -8.0000, A 0.000, B 0.000, C 0.000 }
gfCNCPoint6[2762] = {X 276.2327, Y 102.8800, Z -8.0000, A 0.000, B 0.000, C 0.000 }
gfCNCPoint6[2763] = {X 292.7731, Y 102.8800, Z -8.0000, A 0.000, B 0.000, C 0.000 }
gfCNCPoint6[2764] = {X 293.6844, Y 102.7942, Z -8.0000, A 0.000, B 0.000, C 0.000 }
gfCNCPoint6[2765] = {X 294.5636, Y 102.5397, Z -8.0000, A 0.000, B 0.000, C 0.000 }
gfCNCPoint6[2766] = {X 295.3798, Y 102.1255, Z -8.0000, A 0.000, B 0.000, C 0.000 }
gfCNCPoint6[2767] = {X 296.1043, Y 101.5661, Z -8.0000, A 0.000, B 0.000, C 0.000 }
gfCNCPoint6[2768] = {X 296.7117, Y 100.8813, Z -8.0000, A 0.000, B 0.000, C 0.000 }
gfCNCPoint6[2769] = {X 297.1804, Y 100.0952, Z -8.0000, A 0.000, B 0.000, C 0.000 }
gfCNCPoint6[2770] = {X 319.0966, Y 100.0952, Z -8.0000, A 0.000, B 0.000, C 0.000 }
gfCNCPoint6[2771] = {X 322.1007, Y 101.0514, Z -8.0000, A 0.000, B 0.000, C 0.000 }
gfCNCPoint6[2772] = {X 325.1623, Y 101.8037, Z -8.0000, A 0.000, B 0.000, C 0.000 }
gfCNCPoint6[2773] = {X 328.2675, Y 102.3486, Z -8.0000, A 0.000, B 0.000, C 0.000 }
gfCNCPoint6[2774] = {X 332.9039, Y 102.9207, Z -8.0000, A 0.000, B 0.000, C 0.000 }
gfCNCPoint6[2775] = {X 337.5599, Y 103.3026, Z -8.0000, A 0.000, B 0.000, C 0.000 }
gfCNCPoint6[2776] = {X 342.2276, Y 103.4935, Z -8.0000, A 0.000, B 0.000, C 0.000 }
gfCNCPoint6[2777] = {X 342.3789, Y 103.4959, Z -8.0000, A 0.000, B 0.000, C 0.000 }
gfCNCPoint6[2778] = {X 342.9082, Y 103.5145, Z -8.0000, A 0.000, B 0.000, C 0.000 }
gfCNCPoint6[2779] = {X 349.1744, Y 103.5905, Z -8.0000, A 0.000, B 0.000, C 0.000 }
gfCNCPoint6[2780] = {X 355.4395, Y 103.4514, Z -8.0000, A 0.000, B 0.000, C 0.000 }
gfCNCPoint6[2781] = {X 361.6962, Y 103.0974, Z -8.0000, A 0.000, B 0.000, C 0.000 }
gfCNCPoint6[2782] = {X 365.4559, Y 102.7280, Z -8.0000, A 0.000, B 0.000, C 0.000 }
gfCNCPoint6[2783] = {X 369.1940, Y 102.1818, Z -8.0000, A 0.000, B 0.000, C 0.000 }
gfCNCPoint6[2784] = {X 372.9022, Y 101.4602, Z -8.0000, A 0.000, B 0.000, C 0.000 }
gfCNCPoint6[2785] = {X 375.2305, Y 100.8568, Z -8.0000, A 0.000, B 0.000, C 0.000 }
gfCNCPoint6[2786] = {X 377.5119, Y 100.0952, Z -8.0000, A 0.000, B 0.000, C 0.000 }
gfCNCPoint6[2787] = {X 391.9986, Y 100.0952, Z -8.0000, A 0.000, B 0.000, C 0.000 }
gfCNCPoint6[2788] = {X 392.4674, Y 100.8813, Z -8.0000, A 0.000, B 0.000, C 0.000 }
gfCNCPoint6[2789] = {X 393.0747, Y 101.5661, Z -8.0000, A 0.000, B 0.000, C 0.000 }
gfCNCPoint6[2790] = {X 393.7992, Y 102.1255, Z -8.0000, A 0.000, B 0.000, C 0.000 }
gfCNCPoint6[2791] = {X 394.6155, Y 102.5397, Z -8.0000, A 0.000, B 0.000, C 0.000 }
gfCNCPoint6[2792] = {X 395.4947, Y 102.7942, Z -8.0000, A 0.000, B 0.000, C 0.000 }
gfCNCPoint6[2793] = {X 396.4059, Y 102.8800, Z -8.0000, A 0.000, B 0.000, C 0.000 }
gfCNCPoint6[2794] = {X 415.7067, Y 102.8800, Z -8.0000, A 0.000, B 0.000, C 0.000 }
gfCNCPoint6[2795] = {X 416.6180, Y 102.7942, Z -8.0000, A 0.000, B 0.000, C 0.000 }
gfCNCPoint6[2796] = {X 417.4972, Y 102.5397, Z -8.0000, A 0.000, B 0.000, C 0.000 }
gfCNCPoint6[2797] = {X 418.3134, Y 102.1255, Z -8.0000, A 0.000, B 0.000, C 0.000 }
gfCNCPoint6[2798] = {X 419.0379, Y 101.5661, Z -8.0000, A 0.000, B 0.000, C 0.000 }
gfCNCPoint6[2799] = {X 419.6453, Y 100.8813, Z -8.0000, A 0.000, B 0.000, C 0.000 }
gfCNCPoint6[2800] = {X 420.1140, Y 100.0952, Z -8.0000, A 0.000, B 0.000, C 0.000 }
gfCNCPoint6[2801] = {X 443.7045, Y 100.0952, Z -8.0000, A 0.000, B 0.000, C 0.000 }
gfCNCPoint6[2802] = {X 443.7045, Y 90.4952, Z -8.0000, A 0.000, B 0.000, C 0.000 }
gfCNCPoint6[2803] = {X 448.3230, Y 90.4952, Z -8.0000, A 0.000, B 0.000, C 0.000 }
gfCNCPoint6[2804] = {X 448.4020, Y 90.3748, Z -8.0000, A 0.000, B 0.000, C 0.000 }
gfCNCPoint6[2805] = {X 448.4825, Y 90.2554, Z -8.0000, A 0.000, B 0.000, C 0.000 }
gfCNCPoint6[2806] = {X 445.7365, Y 89.1789, Z -8.0000, A 0.000, B 0.000, C 0.000 }
gfCNCPoint6[2807] = {X 443.7045, Y 90.4952, Z -8.0000, A 0.000, B 0.000, C 0.000 }
gfCNCPoint6[2808] = {X 443.7045, Y 92.8952, Z -8.0000, A 0.000, B 0.000, C 0.000 }
gfCNCPoint6[2809] = {X 449.7242, Y 92.8952, Z -8.0000, A 0.000, B 0.000, C 0.000 }
gfCNCPoint6[2810] = {X 450.0698, Y 92.2376, Z -8.0000, A 0.000, B 0.000, C 0.000 }
gfCNCPoint6[2811] = {X 450.4647, Y 91.6084, Z -8.0000, A 0.000, B 0.000, C 0.000 }
gfCNCPoint6[2812] = {X 451.3969, Y 90.4463, Z -8.0000, A 0.000, B 0.000, C 0.000 }
gfCNCPoint6[2813] = {X 452.4963, Y 89.4409, Z -8.0000, A 0.000, B 0.000, C 0.000 }
gfCNCPoint6[2814] = {X 452.4963, Y 89.2510, Z -8.0000, A 0.000, B 0.000, C 0.000 }
gfCNCPoint6[2815] = {X 445.4655, Y 86.4949, Z -8.0000, A 0.000, B 0.000, C 0.000 }
gfCNCPoint6[2816] = {X 435.5850, Y 92.8952, Z -8.0000, A 0.000, B 0.000, C 0.000 }
gfCNCPoint6[2817] = {X 443.7045, Y 92.8952, Z -8.0000, A 0.000, B 0.000, C 0.000 }
gfCNCPoint6[2818] = {X 443.7045, Y 95.2952, Z -8.0000, A 0.000, B 0.000, C 0.000 }
gfCNCPoint6[2819] = {X 451.3982, Y 95.2952, Z -8.0000, A 0.000, B 0.000, C 0.000 }
gfCNCPoint6[2820] = {X 451.7784, Y 94.1746, Z -8.0000, A 0.000, B 0.000, C 0.000 }
gfCNCPoint6[2821] = {X 452.3351, Y 93.1304, Z -8.0000, A 0.000, B 0.000, C 0.000 }
gfCNCPoint6[2822] = {X 453.0536, Y 92.1901, Z -8.0000, A 0.000, B 0.000, C 0.000 }
gfCNCPoint6[2823] = {X 453.9149, Y 91.3787, Z -8.0000, A 0.000, B 0.000, C 0.000 }
gfCNCPoint6[2824] = {X 454.8963, Y 90.7176, Z -8.0000, A 0.000, B 0.000, C 0.000 }
gfCNCPoint6[2825] = {X 454.8963, Y 87.6139, Z -8.0000, A 0.000, B 0.000, C 0.000 }
gfCNCPoint6[2826] = {X 445.1946, Y 83.8109, Z -8.0000, A 0.000, B 0.000, C 0.000 }
gfCNCPoint6[2827] = {X 427.4656, Y 95.2952, Z -8.0000, A 0.000, B 0.000, C 0.000 }
gfCNCPoint6[2828] = {X 443.7045, Y 95.2952, Z -8.0000, A 0.000, B 0.000, C 0.000 }
gfCNCPoint6[2829] = {X 443.7045, Y 97.6952, Z -8.0000, A 0.000, B 0.000, C 0.000 }
gfCNCPoint6[2830] = {X 453.5796, Y 97.6952, Z -8.0000, A 0.000, B 0.000, C 0.000 }
gfCNCPoint6[2831] = {X 453.5796, Y 97.0659, Z -8.0000, A 0.000, B 0.000, C 0.000 }
gfCNCPoint6[2832] = {X 453.6990, Y 95.9930, Z -8.0000, A 0.000, B 0.000, C 0.000 }
gfCNCPoint6[2833] = {X 454.0514, Y 94.9725, Z -8.0000, A 0.000, B 0.000, C 0.000 }
gfCNCPoint6[2834] = {X 454.6196, Y 94.0545, Z -8.0000, A 0.000, B 0.000, C 0.000 }
gfCNCPoint6[2835] = {X 455.3757, Y 93.2839, Z -8.0000, A 0.000, B 0.000, C 0.000 }
gfCNCPoint6[2836] = {X 456.2827, Y 92.6984, Z -8.0000, A 0.000, B 0.000, C 0.000 }
gfCNCPoint6[2837] = {X 457.2963, Y 92.3266, Z -8.0000, A 0.000, B 0.000, C 0.000 }
gfCNCPoint6[2838] = {X 457.2963, Y 85.9769, Z -8.0000, A 0.000, B 0.000, C 0.000 }
gfCNCPoint6[2839] = {X 444.9237, Y 81.1268, Z -8.0000, A 0.000, B 0.000, C 0.000 }
gfCNCPoint6[2840] = {X 420.5859, Y 96.8921, Z -8.0000, A 0.000, B 0.000, C 0.000 }
gfCNCPoint6[2841] = {X 420.5867, Y 97.0660, Z -8.0000, A 0.000, B 0.000, C 0.000 }
gfCNCPoint6[2842] = {X 420.5867, Y 97.6952, Z -8.0000, A 0.000, B 0.000, C 0.000 }
gfCNCPoint6[2843] = {X 443.7045, Y 97.6952, Z -8.0000, A 0.000, B 0.000, C 0.000 }
gfCNCPoint6[2844] = {X 443.7045, Y 100.0952, Z -8.0000, A 0.000, B 0.000, C 0.000 }
gfCNCPoint6[2845] = {X 454.0523, Y 100.0952, Z -8.0000, A 0.000, B 0.000, C 0.000 }
gfCNCPoint6[2846] = {X 454.5210, Y 100.8813, Z -8.0000, A 0.000, B 0.000, C 0.000 }
gfCNCPoint6[2847] = {X 455.1284, Y 101.5661, Z -8.0000, A 0.000, B 0.000, C 0.000 }
gfCNCPoint6[2848] = {X 455.8529, Y 102.1255, Z -8.0000, A 0.000, B 0.000, C 0.000 }
gfCNCPoint6[2849] = {X 456.6691, Y 102.5397, Z -8.0000, A 0.000, B 0.000, C 0.000 }
gfCNCPoint6[2850] = {X 457.5483, Y 102.7942, Z -8.0000, A 0.000, B 0.000, C 0.000 }
gfCNCPoint6[2851] = {X 458.4596, Y 102.8800, Z -8.0000, A 0.000, B 0.000, C 0.000 }
gfCNCPoint6[2852] = {X 475.0000, Y 102.8800, Z -8.0000, A 0.000, B 0.000, C 0.000 }
gfCNCPoint6[2853] = {X 475.9113, Y 102.7942, Z -8.0000, A 0.000, B 0.000, C 0.000 }
gfCNCPoint6[2854] = {X 476.7905, Y 102.5397, Z -8.0000, A 0.000, B 0.000, C 0.000 }
gfCNCPoint6[2855] = {X 477.6067, Y 102.1255, Z -8.0000, A 0.000, B 0.000, C 0.000 }
gfCNCPoint6[2856] = {X 478.3312, Y 101.5661, Z -8.0000, A 0.000, B 0.000, C 0.000 }
gfCNCPoint6[2857] = {X 478.9386, Y 100.8813, Z -8.0000, A 0.000, B 0.000, C 0.000 }
gfCNCPoint6[2858] = {X 479.4073, Y 100.0952, Z -8.0000, A 0.000, B 0.000, C 0.000 }
gfCNCPoint6[2859] = {X 507.6811, Y 100.0952, Z -8.0000, A 0.000, B 0.000, C 0.000 }
gfCNCPoint6[2860] = {X 507.6811, Y 107.6952, Z -8.0000, A 0.000, B 0.000, C 0.000 }
gfCNCPoint6[2861] = {X 507.6811, Y 107.6952, Z -5.0000, A 0.000, B 0.000, C 0.000 }
gfCNCPoint6[2862] = {X 507.6811, Y 107.6952, Z 11.0000, A 0.000, B 0.000, C 0.000 }
gfCNCPoint6[2863] = {X 108.5573, Y 40.8967, Z 11.0000, A 0.000, B 0.000, C 0.000 }
gfCNCPoint6[2864] = {X 108.5573, Y 40.8967, Z -4.1667, A 0.000, B 0.000, C 0.000 }
gfCNCPoint6[2865] = {X 108.5573, Y 40.8967, Z -8.0000, A 0.000, B 0.000, C 0.000 }
gfCNCPoint6[2866] = {X 108.0701, Y 42.0874, Z -8.0000, A 0.000, B 0.000, C 0.000 }
gfCNCPoint6[2867] = {X 108.0968, Y 42.0409, Z -8.0000, A 0.000, B 0.000, C 0.000 }
gfCNCPoint6[2868] = {X 108.1242, Y 41.9948, Z -8.0000, A 0.000, B 0.000, C 0.000 }
gfCNCPoint6[2869] = {X 108.5476, Y 41.3826, Z -8.0000, A 0.000, B 0.000, C 0.000 }
gfCNCPoint6[2870] = {X 109.0446, Y 40.8286, Z -8.0000, A 0.000, B 0.000, C 0.000 }
gfCNCPoint6[2871] = {X 109.0445, Y 39.7061, Z -8.0000, A 0.000, B 0.000, C 0.000 }
gfCNCPoint6[2872] = {X 108.5573, Y 40.8967, Z -8.0000, A 0.000, B 0.000, C 0.000 }
gfCNCPoint6[2873] = {X 108.5573, Y 40.8967, Z -5.0000, A 0.000, B 0.000, C 0.000 }
gfCNCPoint6[2874] = {X 108.5573, Y 40.8967, Z 11.0000, A 0.000, B 0.000, C 0.000 }
gfCNCPoint6[2875] = {X 95.6819, Y 40.8705, Z 11.0000, A 0.000, B 0.000, C 0.000 }
gfCNCPoint6[2876] = {X 95.6819, Y 40.8705, Z -4.1667, A 0.000, B 0.000, C 0.000 }
gfCNCPoint6[2877] = {X 95.6819, Y 40.8705, Z -8.0000, A 0.000, B 0.000, C 0.000 }
gfCNCPoint6[2878] = {X 95.2123, Y 39.7219, Z -8.0000, A 0.000, B 0.000, C 0.000 }
gfCNCPoint6[2879] = {X 95.2123, Y 40.8680, Z -8.0000, A 0.000, B 0.000, C 0.000 }
gfCNCPoint6[2880] = {X 95.7300, Y 41.4043, Z -8.0000, A 0.000, B 0.000, C 0.000 }
gfCNCPoint6[2881] = {X 96.1516, Y 42.0190, Z -8.0000, A 0.000, B 0.000, C 0.000 }
gfCNCPoint6[2882] = {X 95.6819, Y 40.8705, Z -8.0000, A 0.000, B 0.000, C 0.000 }
gfCNCPoint6[2883] = {X 95.6819, Y 40.8705, Z -5.0000, A 0.000, B 0.000, C 0.000 }
gfCNCPoint6[2884] = {X 95.6819, Y 40.8705, Z 11.0000, A 0.000, B 0.000, C 0.000 }
gfCNCPoint6[2885] = {X -7.6967, Y 43.2782, Z 11.0000, A 0.000, B 0.000, C 0.000 }
gfCNCPoint6[2886] = {X -7.6967, Y 43.2782, Z -5.0000, A 0.000, B 0.000, C 0.000 }
gfCNCPoint6[2887] = {X -7.6967, Y 43.2782, Z -8.0000, A 0.000, B 0.000, C 0.000 }
gfCNCPoint6[2888] = {X -3.6967, Y 30.7976, Z -8.0000, A 0.000, B 0.000, C 0.000 }
gfCNCPoint6[2889] = {X -3.5213, Y 30.2829, Z -8.0000, A 0.000, B 0.000, C 0.000 }
gfCNCPoint6[2890] = {X -3.3272, Y 29.7750, Z -8.0000, A 0.000, B 0.000, C 0.000 }
gfCNCPoint6[2891] = {X -2.7042, Y 28.4548, Z -8.0000, A 0.000, B 0.000, C 0.000 }
gfCNCPoint6[2892] = {X -1.9104, Y 27.2297, Z -8.0000, A 0.000, B 0.000, C 0.000 }
gfCNCPoint6[2893] = {X -0.9601, Y 26.1216, Z -8.0000, A 0.000, B 0.000, C 0.000 }
gfCNCPoint6[2894] = {X 0.1297, Y 25.1503, Z -8.0000, A 0.000, B 0.000, C 0.000 }
gfCNCPoint6[2895] = {X 1.3393, Y 24.3332, Z -8.0000, A 0.000, B 0.000, C 0.000 }
gfCNCPoint6[2896] = {X 0.5792, Y 23.9229, Z -8.0000, A 0.000, B 0.000, C 0.000 }
gfCNCPoint6[2897] = {X -0.0862, Y 23.3720, Z -8.0000, A 0.000, B 0.000, C 0.000 }
gfCNCPoint6[2898] = {X -0.6311, Y 22.7017, Z -8.0000, A 0.000, B 0.000, C 0.000 }
gfCNCPoint6[2899] = {X -1.0345, Y 21.9379, Z -8.0000, A 0.000, B 0.000, C 0.000 }
gfCNCPoint6[2900] = {X -3.6458, Y 15.5423, Z -8.0000, A 0.000, B 0.000, C 0.000 }
gfCNCPoint6[2901] = {X -3.6718, Y 15.4772, Z -8.0000, A 0.000, B 0.000, C 0.000 }
gfCNCPoint6[2902] = {X -3.6967, Y 15.4117, Z -8.0000, A 0.000, B 0.000, C 0.000 }
gfCNCPoint6[2903] = {X -7.6967, Y 4.6466, Z -8.0000, A 0.000, B 0.000, C 0.000 }
gfCNCPoint6[2904] = {X -7.6967, Y 4.6466, Z -5.0000, A 0.000, B 0.000, C 0.000 }
gfCNCPoint6[2905] = {X -7.6967, Y 4.6466, Z 11.0000, A 0.000, B 0.000, C 0.000 }
gfCNCPoint6[2906] = {X -7.6967, Y 16.4131, Z 11.0000, A 0.000, B 0.000, C 0.000 }
gfCNCPoint6[2907] = {X -7.6967, Y 16.4131, Z -5.0000, A 0.000, B 0.000, C 0.000 }
gfCNCPoint6[2908] = {X -7.6967, Y 16.4131, Z -8.0000, A 0.000, B 0.000, C 0.000 }
gfCNCPoint6[2909] = {X -4.8865, Y 16.4131, Z -8.0000, A 0.000, B 0.000, C 0.000 }
gfCNCPoint6[2910] = {X -3.6967, Y 12.5942, Z -8.0000, A 0.000, B 0.000, C 0.000 }
gfCNCPoint6[2911] = {X -3.6607, Y 12.4838, Z -8.0000, A 0.000, B 0.000, C 0.000 }
gfCNCPoint6[2912] = {X -3.6217, Y 12.3744, Z -8.0000, A 0.000, B 0.000, C 0.000 }
gfCNCPoint6[2913] = {X -3.1668, Y 11.4830, Z -8.0000, A 0.000, B 0.000, C 0.000 }
gfCNCPoint6[2914] = {X -2.5189, Y 10.7201, Z -8.0000, A 0.000, B 0.000, C 0.000 }
gfCNCPoint6[2915] = {X -1.7129, Y 10.1268, Z -8.0000, A 0.000, B 0.000, C 0.000 }
gfCNCPoint6[2916] = {X -1.1156, Y 9.7861, Z -8.0000, A 0.000, B 0.000, C 0.000 }
gfCNCPoint6[2917] = {X -0.2329, Y 9.4056, Z -8.0000, A 0.000, B 0.000, C 0.000 }
gfCNCPoint6[2918] = {X 0.7120, Y 9.2298, Z -8.0000, A 0.000, B 0.000, C 0.000 }
gfCNCPoint6[2919] = {X 1.6725, Y 9.2673, Z -8.0000, A 0.000, B 0.000, C 0.000 }
gfCNCPoint6[2920] = {X 2.6009, Y 9.5162, Z -8.0000, A 0.000, B 0.000, C 0.000 }
gfCNCPoint6[2921] = {X 3.4887, Y 9.1191, Z -8.0000, A 0.000, B 0.000, C 0.000 }
gfCNCPoint6[2922] = {X 5.5657, Y 8.3365, Z -8.0000, A 0.000, B 0.000, C 0.000 }
gfCNCPoint6[2923] = {X 7.7065, Y 7.7508, Z -8.0000, A 0.000, B 0.000, C 0.000 }
gfCNCPoint6[2924] = {X 9.8927, Y 7.3671, Z -8.0000, A 0.000, B 0.000, C 0.000 }
gfCNCPoint6[2925] = {X 12.1050, Y 7.1887, Z -8.0000, A 0.000, B 0.000, C 0.000 }
gfCNCPoint6[2926] = {X 14.3244, Y 7.2172, Z -8.0000, A 0.000, B 0.000, C 0.000 }
gfCNCPoint6[2927] = {X 16.5314, Y 7.4523, Z -8.0000, A 0.000, B 0.000, C 0.000 }
gfCNCPoint6[2928] = {X 18.2670, Y 7.8068, Z -8.0000, A 0.000, B 0.000, C 0.000 }
gfCNCPoint6[2929] = {X 19.9576, Y 8.3358, Z -8.0000, A 0.000, B 0.000, C 0.000 }
gfCNCPoint6[2930] = {X 21.5856, Y 9.0340, Z -8.0000, A 0.000, B 0.000, C 0.000 }
gfCNCPoint6[2931] = {X 23.1343, Y 9.8941, Z -8.0000, A 0.000, B 0.000, C 0.000 }
gfCNCPoint6[2932] = {X 24.5875, Y 10.9071, Z -8.0000, A 0.000, B 0.000, C 0.000 }
gfCNCPoint6[2933] = {X 25.6731, Y 11.8564, Z -8.0000, A 0.000, B 0.000, C 0.000 }
gfCNCPoint6[2934] = {X 26.6469, Y 12.9199, Z -8.0000, A 0.000, B 0.000, C 0.000 }
gfCNCPoint6[2935] = {X 27.4970, Y 14.0848, Z -8.0000, A 0.000, B 0.000, C 0.000 }
gfCNCPoint6[2936] = {X 28.2128, Y 15.3366, Z -8.0000, A 0.000, B 0.000, C 0.000 }
gfCNCPoint6[2937] = {X 28.7858, Y 16.6600, Z -8.0000, A 0.000, B 0.000, C 0.000 }
gfCNCPoint6[2938] = {X 29.2603, Y 18.3163, Z -8.0000, A 0.000, B 0.000, C 0.000 }
gfCNCPoint6[2939] = {X 29.5419, Y 20.0160, Z -8.0000, A 0.000, B 0.000, C 0.000 }
gfCNCPoint6[2940] = {X 29.6269, Y 21.7369, Z -8.0000, A 0.000, B 0.000, C 0.000 }
gfCNCPoint6[2941] = {X 29.5141, Y 23.4561, Z -8.0000, A 0.000, B 0.000, C 0.000 }
gfCNCPoint6[2942] = {X 29.2050, Y 25.1511, Z -8.0000, A 0.000, B 0.000, C 0.000 }
gfCNCPoint6[2943] = {X 28.7623, Y 26.5973, Z -8.0000, A 0.000, B 0.000, C 0.000 }
gfCNCPoint6[2944] = {X 28.1368, Y 27.9742, Z -8.0000, A 0.000, B 0.000, C 0.000 }
gfCNCPoint6[2945] = {X 27.3389, Y 29.2590, Z -8.0000, A 0.000, B 0.000, C 0.000 }
gfCNCPoint6[2946] = {X 26.3819, Y 30.4300, Z -8.0000, A 0.000, B 0.000, C 0.000 }
gfCNCPoint6[2947] = {X 25.2819, Y 31.4679, Z -8.0000, A 0.000, B 0.000, C 0.000 }
gfCNCPoint6[2948] = {X 26.0857, Y 31.8100, Z -8.0000, A 0.000, B 0.000, C 0.000 }
gfCNCPoint6[2949] = {X 26.8042, Y 32.3069, Z -8.0000, A 0.000, B 0.000, C 0.000 }
gfCNCPoint6[2950] = {X 27.4081, Y 32.9382, Z -8.0000, A 0.000, B 0.000, C 0.000 }
gfCNCPoint6[2951] = {X 27.8726, Y 33.6781, Z -8.0000, A 0.000, B 0.000, C 0.000 }
gfCNCPoint6[2952] = {X 30.9100, Y 39.9530, Z -8.0000, A 0.000, B 0.000, C 0.000 }
gfCNCPoint6[2953] = {X 31.2306, Y 40.8622, Z -8.0000, A 0.000, B 0.000, C 0.000 }
gfCNCPoint6[2954] = {X 31.3415, Y 41.8197, Z -8.0000, A 0.000, B 0.000, C 0.000 }
gfCNCPoint6[2955] = {X 31.2374, Y 42.7781, Z -8.0000, A 0.000, B 0.000, C 0.000 }
gfCNCPoint6[2956] = {X 30.9234, Y 43.6895, Z -8.0000, A 0.000, B 0.000, C 0.000 }
gfCNCPoint6[2957] = {X 30.4150, Y 44.5085, Z -8.0000, A 0.000, B 0.000, C 0.000 }
gfCNCPoint6[2958] = {X 29.7377, Y 45.1945, Z -8.0000, A 0.000, B 0.000, C 0.000 }
gfCNCPoint6[2959] = {X 29.2018, Y 45.6278, Z -8.0000, A 0.000, B 0.000, C 0.000 }
gfCNCPoint6[2960] = {X 28.4981, Y 46.0917, Z -8.0000, A 0.000, B 0.000, C 0.000 }
gfCNCPoint6[2961] = {X 27.7179, Y 46.4105, Z -8.0000, A 0.000, B 0.000, C 0.000 }
gfCNCPoint6[2962] = {X 26.8907, Y 46.5721, Z -8.0000, A 0.000, B 0.000, C 0.000 }
gfCNCPoint6[2963] = {X 26.0479, Y 46.5704, Z -8.0000, A 0.000, B 0.000, C 0.000 }
gfCNCPoint6[2964] = {X 25.2214, Y 46.4054, Z -8.0000, A 0.000, B 0.000, C 0.000 }
gfCNCPoint6[2965] = {X 23.4208, Y 47.3544, Z -8.0000, A 0.000, B 0.000, C 0.000 }
gfCNCPoint6[2966] = {X 21.5588, Y 48.1767, Z -8.0000, A 0.000, B 0.000, C 0.000 }
gfCNCPoint6[2967] = {X 19.6445, Y 48.8683, Z -8.0000, A 0.000, B 0.000, C 0.000 }
gfCNCPoint6[2968] = {X 17.7046, Y 49.4160, Z -8.0000, A 0.000, B 0.000, C 0.000 }
gfCNCPoint6[2969] = {X 15.7237, Y 49.7899, Z -8.0000, A 0.000, B 0.000, C 0.000 }
gfCNCPoint6[2970] = {X 13.7175, Y 49.9870, Z -8.0000, A 0.000, B 0.000, C 0.000 }
gfCNCPoint6[2971] = {X 11.7018, Y 50.0057, Z -8.0000, A 0.000, B 0.000, C 0.000 }
gfCNCPoint6[2972] = {X 9.6923, Y 49.8460, Z -8.0000, A 0.000, B 0.000, C 0.000 }
gfCNCPoint6[2973] = {X 7.7049, Y 49.5090, Z -8.0000, A 0.000, B 0.000, C 0.000 }
gfCNCPoint6[2974] = {X 5.8033, Y 48.9880, Z -8.0000, A 0.000, B 0.000, C 0.000 }
gfCNCPoint6[2975] = {X 3.9763, Y 48.2468, Z -8.0000, A 0.000, B 0.000, C 0.000 }
gfCNCPoint6[2976] = {X 2.2493, Y 47.2955, Z -8.0000, A 0.000, B 0.000, C 0.000 }
gfCNCPoint6[2977] = {X 0.6463, Y 46.1475, Z -8.0000, A 0.000, B 0.000, C 0.000 }
gfCNCPoint6[2978] = {X -0.4855, Y 45.1297, Z -8.0000, A 0.000, B 0.000, C 0.000 }
gfCNCPoint6[2979] = {X -1.4909, Y 43.9868, Z -8.0000, A 0.000, B 0.000, C 0.000 }
gfCNCPoint6[2980] = {X -2.3560, Y 42.7344, Z -8.0000, A 0.000, B 0.000, C 0.000 }
gfCNCPoint6[2981] = {X -3.0692, Y 41.3897, Z -8.0000, A 0.000, B 0.000, C 0.000 }
gfCNCPoint6[2982] = {X -3.6206, Y 39.9709, Z -8.0000, A 0.000, B 0.000, C 0.000 }
gfCNCPoint6[2983] = {X -3.6592, Y 39.8491, Z -8.0000, A 0.000, B 0.000, C 0.000 }
gfCNCPoint6[2984] = {X -3.6967, Y 39.7269, Z -8.0000, A 0.000, B 0.000, C 0.000 }
gfCNCPoint6[2985] = {X -4.8504, Y 35.8969, Z -8.0000, A 0.000, B 0.000, C 0.000 }
gfCNCPoint6[2986] = {X -7.9953, Y 36.0104, Z -8.0000, A 0.000, B 0.000, C 0.000 }
gfCNCPoint6[2987] = {X -7.9953, Y 36.0104, Z -5.0000, A 0.000, B 0.000, C 0.000 }
gfCNCPoint6[2988] = {X -7.9953, Y 36.0104, Z 11.0000, A 0.000, B 0.000, C 0.000 }
gfCNCPoint6[2989] = {X 608.0000, Y 40.1188, Z 11.0000, A 0.000, B 0.000, C 0.000 }
gfCNCPoint6[2990] = {X 608.0000, Y 40.1188, Z -5.0000, A 0.000, B 0.000, C 0.000 }
gfCNCPoint6[2991] = {X 608.0000, Y 40.1188, Z -8.0000, A 0.000, B 0.000, C 0.000 }
gfCNCPoint6[2992] = {X 603.6967, Y 47.2354, Z -8.0000, A 0.000, B 0.000, C 0.000 }
gfCNCPoint6[2993] = {X 603.6635, Y 47.2894, Z -8.0000, A 0.000, B 0.000, C 0.000 }
gfCNCPoint6[2994] = {X 603.6295, Y 47.3429, Z -8.0000, A 0.000, B 0.000, C 0.000 }
gfCNCPoint6[2995] = {X 603.0931, Y 48.0158, Z -8.0000, A 0.000, B 0.000, C 0.000 }
gfCNCPoint6[2996] = {X 602.4341, Y 48.5690, Z -8.0000, A 0.000, B 0.000, C 0.000 }
gfCNCPoint6[2997] = {X 601.6784, Y 48.9806, Z -8.0000, A 0.000, B 0.000, C 0.000 }
gfCNCPoint6[2998] = {X 600.8562, Y 49.2343, Z -8.0000, A 0.000, B 0.000, C 0.000 }
gfCNCPoint6[2999] = {X 600.0000, Y 49.3200, Z -8.0000, A 0.000, B 0.000, C 0.000 }
gfCNCPoint6[3000] = {X 593.5565, Y 49.3200, Z -8.0000, A 0.000, B 0.000, C 0.000 }
gfCNCPoint6[3001] = {X 592.5952, Y 49.2117, Z -8.0000, A 0.000, B 0.000, C 0.000 }
gfCNCPoint6[3002] = {X 591.6822, Y 48.8922, Z -8.0000, A 0.000, B 0.000, C 0.000 }
gfCNCPoint6[3003] = {X 590.8631, Y 48.3775, Z -8.0000, A 0.000, B 0.000, C 0.000 }
gfCNCPoint6[3004] = {X 590.1790, Y 47.6935, Z -8.0000, A 0.000, B 0.000, C 0.000 }
gfCNCPoint6[3005] = {X 589.6643, Y 46.8744, Z -8.0000, A 0.000, B 0.000, C 0.000 }
gfCNCPoint6[3006] = {X 589.3448, Y 45.9613, Z -8.0000, A 0.000, B 0.000, C 0.000 }
gfCNCPoint6[3007] = {X 589.2365, Y 45.0000, Z -8.0000, A 0.000, B 0.000, C 0.000 }
gfCNCPoint6[3008] = {X 589.2365, Y 44.0648, Z -8.0000, A 0.000, B 0.000, C 0.000 }
gfCNCPoint6[3009] = {X 589.3401, Y 43.1364, Z -8.0000, A 0.000, B 0.000, C 0.000 }
gfCNCPoint6[3010] = {X 589.6393, Y 42.2514, Z -8.0000, A 0.000, B 0.000, C 0.000 }
gfCNCPoint6[3011] = {X 590.1202, Y 41.4506, Z -8.0000, A 0.000, B 0.000, C 0.000 }
gfCNCPoint6[3012] = {X 590.7609, Y 40.7707, Z -8.0000, A 0.000, B 0.000, C 0.000 }
gfCNCPoint6[3013] = {X 590.7617, Y 33.5335, Z -8.0000, A 0.000, B 0.000, C 0.000 }
gfCNCPoint6[3014] = {X 585.4453, Y 46.6524, Z -8.0000, A 0.000, B 0.000, C 0.000 }
gfCNCPoint6[3015] = {X 585.0755, Y 47.3550, Z -8.0000, A 0.000, B 0.000, C 0.000 }
gfCNCPoint6[3016] = {X 584.5834, Y 47.9780, Z -8.0000, A 0.000, B 0.000, C 0.000 }
gfCNCPoint6[3017] = {X 583.9856, Y 48.5004, Z -8.0000, A 0.000, B 0.000, C 0.000 }
gfCNCPoint6[3018] = {X 583.3023, Y 48.9046, Z -8.0000, A 0.000, B 0.000, C 0.000 }
gfCNCPoint6[3019] = {X 582.3585, Y 49.2242, Z -8.0000, A 0.000, B 0.000, C 0.000 }
gfCNCPoint6[3020] = {X 581.3666, Y 49.3191, Z -8.0000, A 0.000, B 0.000, C 0.000 }
gfCNCPoint6[3021] = {X 580.3794, Y 49.1842, Z -8.0000, A 0.000, B 0.000, C 0.000 }
gfCNCPoint6[3022] = {X 579.4493, Y 48.8268, Z -8.0000, A 0.000, B 0.000, C 0.000 }
gfCNCPoint6[3023] = {X 578.6259, Y 48.2657, Z -8.0000, A 0.000, B 0.000, C 0.000 }
gfCNCPoint6[3024] = {X 577.9529, Y 47.5309, Z -8.0000, A 0.000, B 0.000, C 0.000 }
gfCNCPoint6[3025] = {X 577.4662, Y 46.6615, Z -8.0000, A 0.000, B 0.000, C 0.000 }
gfCNCPoint6[3026] = {X 572.0202, Y 33.3448, Z -8.0000, A 0.000, B 0.000, C 0.000 }
gfCNCPoint6[3027] = {X 572.0204, Y 40.7711, Z -8.0000, A 0.000, B 0.000, C 0.000 }
gfCNCPoint6[3028] = {X 572.6583, Y 41.4421, Z -8.0000, A 0.000, B 0.000, C 0.000 }
gfCNCPoint6[3029] = {X 573.1385, Y 42.2336, Z -8.0000, A 0.000, B 0.000, C 0.000 }
gfCNCPoint6[3030] = {X 573.4391, Y 43.1092, Z -8.0000, A 0.000, B 0.000, C 0.000 }
gfCNCPoint6[3031] = {X 573.5463, Y 44.0287, Z -8.0000, A 0.000, B 0.000, C 0.000 }
gfCNCPoint6[3032] = {X 573.5464, Y 45.0000, Z -8.0000, A 0.000, B 0.000, C 0.000 }
gfCNCPoint6[3033] = {X 573.4381, Y 45.9613, Z -8.0000, A 0.000, B 0.000, C 0.000 }
gfCNCPoint6[3034] = {X 573.1186, Y 46.8744, Z -8.0000, A 0.000, B 0.000, C 0.000 }
gfCNCPoint6[3035] = {X 572.6039, Y 47.6935, Z -8.0000, A 0.000, B 0.000, C 0.000 }
gfCNCPoint6[3036] = {X 571.9199, Y 48.3775, Z -8.0000, A 0.000, B 0.000, C 0.000 }
gfCNCPoint6[3037] = {X 571.1008, Y 48.8922, Z -8.0000, A 0.000, B 0.000, C 0.000 }
gfCNCPoint6[3038] = {X 570.1877, Y 49.2117, Z -8.0000, A 0.000, B 0.000, C 0.000 }
gfCNCPoint6[3039] = {X 569.2264, Y 49.3200, Z -8.0000, A 0.000, B 0.000, C 0.000 }
gfCNCPoint6[3040] = {X 562.4443, Y 49.3200, Z -8.0000, A 0.000, B 0.000, C 0.000 }
gfCNCPoint6[3041] = {X 561.4830, Y 49.2117, Z -8.0000, A 0.000, B 0.000, C 0.000 }
gfCNCPoint6[3042] = {X 560.5699, Y 48.8922, Z -8.0000, A 0.000, B 0.000, C 0.000 }
gfCNCPoint6[3043] = {X 559.7508, Y 48.3775, Z -8.0000, A 0.000, B 0.000, C 0.000 }
gfCNCPoint6[3044] = {X 559.0668, Y 47.6935, Z -8.0000, A 0.000, B 0.000, C 0.000 }
gfCNCPoint6[3045] = {X 558.5521, Y 46.8744, Z -8.0000, A 0.000, B 0.000, C 0.000 }
gfCNCPoint6[3046] = {X 558.2326, Y 45.9613, Z -8.0000, A 0.000, B 0.000, C 0.000 }
gfCNCPoint6[3047] = {X 558.1243, Y 45.0000, Z -8.0000, A 0.000, B 0.000, C 0.000 }
gfCNCPoint6[3048] = {X 558.1243, Y 44.0650, Z -8.0000, A 0.000, B 0.000, C 0.000 }
gfCNCPoint6[3049] = {X 558.2277, Y 43.1361, Z -8.0000, A 0.000, B 0.000, C 0.000 }
gfCNCPoint6[3050] = {X 558.5271, Y 42.2507, Z -8.0000, A 0.000, B 0.000, C 0.000 }
gfCNCPoint6[3051] = {X 559.0088, Y 41.4498, Z -8.0000, A 0.000, B 0.000, C 0.000 }
gfCNCPoint6[3052] = {X 559.6506, Y 40.7703, Z -8.0000, A 0.000, B 0.000, C 0.000 }
gfCNCPoint6[3053] = {X 559.6510, Y 9.2295, Z -8.0000, A 0.000, B 0.000, C 0.000 }
gfCNCPoint6[3054] = {X 559.0129, Y 8.5586, Z -8.0000, A 0.000, B 0.000, C 0.000 }
gfCNCPoint6[3055] = {X 558.5325, Y 7.7671, Z -8.0000, A 0.000, B 0.000, C 0.000 }
gfCNCPoint6[3056] = {X 558.2317, Y 6.8915, Z -8.0000, A 0.000, B 0.000, C 0.000 }
gfCNCPoint6[3057] = {X 558.1245, Y 5.9718, Z -8.0000, A 0.000, B 0.000, C 0.000 }
gfCNCPoint6[3058] = {X 558.1243, Y 5.0000, Z -8.0000, A 0.000, B 0.000, C 0.000 }
gfCNCPoint6[3059] = {X 558.2326, Y 4.0387, Z -8.0000, A 0.000, B 0.000, C 0.000 }
gfCNCPoint6[3060] = {X 558.5521, Y 3.1256, Z -8.0000, A 0.000, B 0.000, C 0.000 }
gfCNCPoint6[3061] = {X 559.0668, Y 2.3065, Z -8.0000, A 0.000, B 0.000, C 0.000 }
gfCNCPoint6[3062] = {X 559.7508, Y 1.6225, Z -8.0000, A 0.000, B 0.000, C 0.000 }
gfCNCPoint6[3063] = {X 560.5699, Y 1.1078, Z -8.0000, A 0.000, B 0.000, C 0.000 }
gfCNCPoint6[3064] = {X 561.4830, Y 0.7883, Z -8.0000, A 0.000, B 0.000, C 0.000 }
gfCNCPoint6[3065] = {X 562.4443, Y 0.6800, Z -8.0000, A 0.000, B 0.000, C 0.000 }
gfCNCPoint6[3066] = {X 570.9376, Y 0.6800, Z -8.0000, A 0.000, B 0.000, C 0.000 }
gfCNCPoint6[3067] = {X 571.8988, Y 0.7883, Z -8.0000, A 0.000, B 0.000, C 0.000 }
gfCNCPoint6[3068] = {X 572.8119, Y 1.1078, Z -8.0000, A 0.000, B 0.000, C 0.000 }
gfCNCPoint6[3069] = {X 573.6310, Y 1.6225, Z -8.0000, A 0.000, B 0.000, C 0.000 }
gfCNCPoint6[3070] = {X 574.3151, Y 2.3065, Z -8.0000, A 0.000, B 0.000, C 0.000 }
gfCNCPoint6[3071] = {X 574.8297, Y 3.1256, Z -8.0000, A 0.000, B 0.000, C 0.000 }
gfCNCPoint6[3072] = {X 575.1492, Y 4.0387, Z -8.0000, A 0.000, B 0.000, C 0.000 }
gfCNCPoint6[3073] = {X 575.2576, Y 5.0000, Z -8.0000, A 0.000, B 0.000, C 0.000 }
gfCNCPoint6[3074] = {X 575.2576, Y 5.9343, Z -8.0000, A 0.000, B 0.000, C 0.000 }
gfCNCPoint6[3075] = {X 575.1836, Y 6.7301, Z -8.0000, A 0.000, B 0.000, C 0.000 }
gfCNCPoint6[3076] = {X 574.9643, Y 7.4986, Z -8.0000, A 0.000, B 0.000, C 0.000 }
gfCNCPoint6[3077] = {X 574.6072, Y 8.2136, Z -8.0000, A 0.000, B 0.000, C 0.000 }
gfCNCPoint6[3078] = {X 581.1910, Y 24.3685, Z -8.0000, A 0.000, B 0.000, C 0.000 }
gfCNCPoint6[3079] = {X 587.8454, Y 8.0936, Z -8.0000, A 0.000, B 0.000, C 0.000 }
gfCNCPoint6[3080] = {X 587.5315, Y 7.4226, Z -8.0000, A 0.000, B 0.000, C 0.000 }
gfCNCPoint6[3081] = {X 587.3368, Y 6.7080, Z -8.0000, A 0.000, B 0.000, C 0.000 }
gfCNCPoint6[3082] = {X 587.2671, Y 5.9705, Z -8.0000, A 0.000, B 0.000, C 0.000 }
gfCNCPoint6[3083] = {X 587.2670, Y 5.0000, Z -8.0000, A 0.000, B 0.000, C 0.000 }
gfCNCPoint6[3084] = {X 587.3753, Y 4.0387, Z -8.0000, A 0.000, B 0.000, C 0.000 }
gfCNCPoint6[3085] = {X 587.6948, Y 3.1256, Z -8.0000, A 0.000, B 0.000, C 0.000 }
gfCNCPoint6[3086] = {X 588.2094, Y 2.3065, Z -8.0000, A 0.000, B 0.000, C 0.000 }
gfCNCPoint6[3087] = {X 588.8935, Y 1.6225, Z -8.0000, A 0.000, B 0.000, C 0.000 }
gfCNCPoint6[3088] = {X 589.7126, Y 1.1078, Z -8.0000, A 0.000, B 0.000, C 0.000 }
gfCNCPoint6[3089] = {X 590.6257, Y 0.7883, Z -8.0000, A 0.000, B 0.000, C 0.000 }
gfCNCPoint6[3090] = {X 591.5870, Y 0.6800, Z -8.0000, A 0.000, B 0.000, C 0.000 }
gfCNCPoint6[3091] = {X 600.0000, Y 0.6800, Z -8.0000, A 0.000, B 0.000, C 0.000 }
gfCNCPoint6[3092] = {X 600.8562, Y 0.7657, Z -8.0000, A 0.000, B 0.000, C 0.000 }
gfCNCPoint6[3093] = {X 601.6784, Y 1.0194, Z -8.0000, A 0.000, B 0.000, C 0.000 }
gfCNCPoint6[3094] = {X 602.4341, Y 1.4310, Z -8.0000, A 0.000, B 0.000, C 0.000 }
gfCNCPoint6[3095] = {X 603.0931, Y 1.9842, Z -8.0000, A 0.000, B 0.000, C 0.000 }
gfCNCPoint6[3096] = {X 603.6295, Y 2.6571, Z -8.0000, A 0.000, B 0.000, C 0.000 }
gfCNCPoint6[3097] = {X 603.6635, Y 2.7106, Z -8.0000, A 0.000, B 0.000, C 0.000 }
gfCNCPoint6[3098] = {X 603.6967, Y 2.7646, Z -8.0000, A 0.000, B 0.000, C 0.000 }
gfCNCPoint6[3099] = {X 608.0000, Y 9.8812, Z -8.0000, A 0.000, B 0.000, C 0.000 }
gfCNCPoint6[3100] = {X 608.0000, Y 9.8812, Z -5.0000, A 0.000, B 0.000, C 0.000 }
gfCNCPoint6[3101] = {X 608.0000, Y 9.8812, Z 11.0000, A 0.000, B 0.000, C 0.000 }
gfCNCPoint6[3102] = {X -7.6967, Y 16.7871, Z 11.0000, A 0.000, B 0.000, C 0.000 }
gfCNCPoint6[3103] = {X -7.6967, Y 16.7871, Z -5.0000, A 0.000, B 0.000, C 0.000 }
gfCNCPoint6[3104] = {X -7.6967, Y 16.7871, Z -8.0000, A 0.000, B 0.000, C 0.000 }
gfCNCPoint6[3105] = {X -4.6241, Y 16.7871, Z -8.0000, A 0.000, B 0.000, C 0.000 }
gfCNCPoint6[3106] = {X -3.6967, Y 12.8961, Z -8.0000, A 0.000, B 0.000, C 0.000 }
gfCNCPoint6[3107] = {X -3.6292, Y 12.6469, Z -8.0000, A 0.000, B 0.000, C 0.000 }
gfCNCPoint6[3108] = {X -3.5467, Y 12.4023, Z -8.0000, A 0.000, B 0.000, C 0.000 }
gfCNCPoint6[3109] = {X -3.1002, Y 11.5274, Z -8.0000, A 0.000, B 0.000, C 0.000 }
gfCNCPoint6[3110] = {X -2.4644, Y 10.7786, Z -8.0000, A 0.000, B 0.000, C 0.000 }
gfCNCPoint6[3111] = {X -1.6733, Y 10.1963, Z -8.0000, A 0.000, B 0.000, C 0.000 }
gfCNCPoint6[3112] = {X -1.0760, Y 9.8555, Z -8.0000, A 0.000, B 0.000, C 0.000 }
gfCNCPoint6[3113] = {X -0.2016, Y 9.4797, Z -8.0000, A 0.000, B 0.000, C 0.000 }
gfCNCPoint6[3114] = {X 0.7345, Y 9.3084, Z -8.0000, A 0.000, B 0.000, C 0.000 }
gfCNCPoint6[3115] = {X 1.6853, Y 9.3502, Z -8.0000, A 0.000, B 0.000, C 0.000 }
gfCNCPoint6[3116] = {X 2.6028, Y 9.6030, Z -8.0000, A 0.000, B 0.000, C 0.000 }
gfCNCPoint6[3117] = {X 3.5209, Y 9.1923, Z -8.0000, A 0.000, B 0.000, C 0.000 }
gfCNCPoint6[3118] = {X 5.5908, Y 8.4124, Z -8.0000, A 0.000, B 0.000, C 0.000 }
gfCNCPoint6[3119] = {X 7.7244, Y 7.8288, Z -8.0000, A 0.000, B 0.000, C 0.000 }
gfCNCPoint6[3120] = {X 9.9031, Y 7.4464, Z -8.0000, A 0.000, B 0.000, C 0.000 }
gfCNCPoint6[3121] = {X 12.1079, Y 7.2686, Z -8.0000, A 0.000, B 0.000, C 0.000 }
gfCNCPoint6[3122] = {X 14.3197, Y 7.2970, Z -8.0000, A 0.000, B 0.000, C 0.000 }
gfCNCPoint6[3123] = {X 16.5192, Y 7.5313, Z -8.0000, A 0.000, B 0.000, C 0.000 }
gfCNCPoint6[3124] = {X 18.2469, Y 7.8842, Z -8.0000, A 0.000, B 0.000, C 0.000 }
gfCNCPoint6[3125] = {X 19.9298, Y 8.4108, Z -8.0000, A 0.000, B 0.000, C 0.000 }
gfCNCPoint6[3126] = {X 21.5504, Y 9.1058, Z -8.0000, A 0.000, B 0.000, C 0.000 }
gfCNCPoint6[3127] = {X 23.0919, Y 9.9620, Z -8.0000, A 0.000, B 0.000, C 0.000 }
gfCNCPoint6[3128] = {X 24.5385, Y 10.9703, Z -8.0000, A 0.000, B 0.000, C 0.000 }
gfCNCPoint6[3129] = {X 25.6173, Y 11.9137, Z -8.0000, A 0.000, B 0.000, C 0.000 }
gfCNCPoint6[3130] = {X 26.5851, Y 12.9707, Z -8.0000, A 0.000, B 0.000, C 0.000 }
gfCNCPoint6[3131] = {X 27.4299, Y 14.1284, Z -8.0000, A 0.000, B 0.000, C 0.000 }
gfCNCPoint6[3132] = {X 28.1413, Y 15.3725, Z -8.0000, A 0.000, B 0.000, C 0.000 }
gfCNCPoint6[3133] = {X 28.7107, Y 16.6876, Z -8.0000, A 0.000, B 0.000, C 0.000 }
gfCNCPoint6[3134] = {X 29.1825, Y 18.3349, Z -8.0000, A 0.000, B 0.000, C 0.000 }
gfCNCPoint6[3135] = {X 29.4625, Y 20.0255, Z -8.0000, A 0.000, B 0.000, C 0.000 }
gfCNCPoint6[3136] = {X 29.5469, Y 21.7369, Z -8.0000, A 0.000, B 0.000, C 0.000 }
gfCNCPoint6[3137] = {X 29.4346, Y 23.4468, Z -8.0000, A 0.000, B 0.000, C 0.000 }
gfCNCPoint6[3138] = {X 29.1272, Y 25.1325, Z -8.0000, A 0.000, B 0.000, C 0.000 }
gfCNCPoint6[3139] = {X 28.6768, Y 26.5971, Z -8.0000, A 0.000, B 0.000, C 0.000 }
gfCNCPoint6[3140] = {X 28.0376, Y 27.9898, Z -8.0000, A 0.000, B 0.000, C 0.000 }
gfCNCPoint6[3141] = {X 27.2207, Y 29.2862, Z -8.0000, A 0.000, B 0.000, C 0.000 }
gfCNCPoint6[3142] = {X 26.2403, Y 30.4638, Z -8.0000, A 0.000, B 0.000, C 0.000 }
gfCNCPoint6[3143] = {X 25.1135, Y 31.5021, Z -8.0000, A 0.000, B 0.000, C 0.000 }
gfCNCPoint6[3144] = {X 25.2530, Y 31.5427, Z -8.0000, A 0.000, B 0.000, C 0.000 }
gfCNCPoint6[3145] = {X 25.3910, Y 31.5879, Z -8.0000, A 0.000, B 0.000, C 0.000 }
gfCNCPoint6[3146] = {X 26.1383, Y 31.9319, Z -8.0000, A 0.000, B 0.000, C 0.000 }
gfCNCPoint6[3147] = {X 26.8051, Y 32.4136, Z -8.0000, A 0.000, B 0.000, C 0.000 }
gfCNCPoint6[3148] = {X 27.3663, Y 33.0151, Z -8.0000, A 0.000, B 0.000, C 0.000 }
gfCNCPoint6[3149] = {X 27.8009, Y 33.7136, Z -8.0000, A 0.000, B 0.000, C 0.000 }
gfCNCPoint6[3150] = {X 30.8380, Y 39.9879, Z -8.0000, A 0.000, B 0.000, C 0.000 }
gfCNCPoint6[3151] = {X 31.1526, Y 40.8802, Z -8.0000, A 0.000, B 0.000, C 0.000 }
gfCNCPoint6[3152] = {X 31.2615, Y 41.8200, Z -8.0000, A 0.000, B 0.000, C 0.000 }
gfCNCPoint6[3153] = {X 31.1593, Y 42.7606, Z -8.0000, A 0.000, B 0.000, C 0.000 }
gfCNCPoint6[3154] = {X 30.8511, Y 43.6551, Z -8.0000, A 0.000, B 0.000, C 0.000 }
gfCNCPoint6[3155] = {X 30.3522, Y 44.4590, Z -8.0000, A 0.000, B 0.000, C 0.000 }
gfCNCPoint6[3156] = {X 29.6874, Y 45.1323, Z -8.0000, A 0.000, B 0.000, C 0.000 }
gfCNCPoint6[3157] = {X 29.1514, Y 45.5656, Z -8.0000, A 0.000, B 0.000, C 0.000 }
gfCNCPoint6[3158] = {X 28.4547, Y 46.0242, Z -8.0000, A 0.000, B 0.000, C 0.000 }
gfCNCPoint6[3159] = {X 27.6818, Y 46.3378, Z -8.0000, A 0.000, B 0.000, C 0.000 }
gfCNCPoint6[3160] = {X 26.8625, Y 46.4944, Z -8.0000, A 0.000, B 0.000, C 0.000 }
gfCNCPoint6[3161] = {X 26.0285, Y 46.4880, Z -8.0000, A 0.000, B 0.000, C 0.000 }
gfCNCPoint6[3162] = {X 25.2117, Y 46.3187, Z -8.0000, A 0.000, B 0.000, C 0.000 }
gfCNCPoint6[3163] = {X 23.4066, Y 47.2724, Z -8.0000, A 0.000, B 0.000, C 0.000 }
gfCNCPoint6[3164] = {X 21.5396, Y 48.0982, Z -8.0000, A 0.000, B 0.000, C 0.000 }
gfCNCPoint6[3165] = {X 19.6197, Y 48.7922, Z -8.0000, A 0.000, B 0.000, C 0.000 }
gfCNCPoint6[3166] = {X 17.6864, Y 49.3381, Z -8.0000, A 0.000, B 0.000, C 0.000 }
gfCNCPoint6[3167] = {X 15.7125, Y 49.7107, Z -8.0000, A 0.000, B 0.000, C 0.000 }
gfCNCPoint6[3168] = {X 13.7133, Y 49.9071, Z -8.0000, A 0.000, B 0.000, C 0.000 }
gfCNCPoint6[3169] = {X 11.7046, Y 49.9258, Z -8.0000, A 0.000, B 0.000, C 0.000 }
gfCNCPoint6[3170] = {X 9.7021, Y 49.7666, Z -8.0000, A 0.000, B 0.000, C 0.000 }
gfCNCPoint6[3171] = {X 7.7216, Y 49.4307, Z -8.0000, A 0.000, B 0.000, C 0.000 }
gfCNCPoint6[3172] = {X 5.8290, Y 48.9123, Z -8.0000, A 0.000, B 0.000, C 0.000 }
gfCNCPoint6[3173] = {X 4.0106, Y 48.1745, Z -8.0000, A 0.000, B 0.000, C 0.000 }
gfCNCPoint6[3174] = {X 2.2918, Y 47.2278, Z -8.0000, A 0.000, B 0.000, C 0.000 }
gfCNCPoint6[3175] = {X 0.6965, Y 46.0852, Z -8.0000, A 0.000, B 0.000, C 0.000 }
gfCNCPoint6[3176] = {X -0.4285, Y 45.0736, Z -8.0000, A 0.000, B 0.000, C 0.000 }
gfCNCPoint6[3177] = {X -1.4277, Y 43.9377, Z -8.0000, A 0.000, B 0.000, C 0.000 }
gfCNCPoint6[3178] = {X -2.2876, Y 42.6930, Z -8.0000, A 0.000, B 0.000, C 0.000 }
gfCNCPoint6[3179] = {X -2.9964, Y 41.3565, Z -8.0000, A 0.000, B 0.000, C 0.000 }
gfCNCPoint6[3180] = {X -3.5444, Y 39.9463, Z -8.0000, A 0.000, B 0.000, C 0.000 }
gfCNCPoint6[3181] = {X -3.6232, Y 39.6936, Z -8.0000, A 0.000, B 0.000, C 0.000 }
gfCNCPoint6[3182] = {X -3.6967, Y 39.4393, Z -8.0000, A 0.000, B 0.000, C 0.000 }
gfCNCPoint6[3183] = {X -4.7687, Y 35.5857, Z -8.0000, A 0.000, B 0.000, C 0.000 }
gfCNCPoint6[3184] = {X -8.0050, Y 35.6371, Z -8.0000, A 0.000, B 0.000, C 0.000 }
gfCNCPoint6[3185] = {X -8.0050, Y 35.6371, Z -5.0000, A 0.000, B 0.000, C 0.000 }
gfCNCPoint6[3186] = {X -8.0050, Y 35.6371, Z 11.0000, A 0.000, B 0.000, C 0.000 }
gfCNCPoint6[3187] = {X -7.6967, Y 17.3025, Z 11.0000, A 0.000, B 0.000, C 0.000 }
gfCNCPoint6[3188] = {X -7.6967, Y 17.3025, Z -5.0000, A 0.000, B 0.000, C 0.000 }
gfCNCPoint6[3189] = {X -7.6967, Y 17.3025, Z -8.0000, A 0.000, B 0.000, C 0.000 }
gfCNCPoint6[3190] = {X -4.2183, Y 17.3025, Z -8.0000, A 0.000, B 0.000, C 0.000 }
gfCNCPoint6[3191] = {X -3.6967, Y 13.3366, Z -8.0000, A 0.000, B 0.000, C 0.000 }
gfCNCPoint6[3192] = {X -3.6097, Y 12.8771, Z -8.0000, A 0.000, B 0.000, C 0.000 }
gfCNCPoint6[3193] = {X -3.4717, Y 12.4302, Z -8.0000, A 0.000, B 0.000, C 0.000 }
gfCNCPoint6[3194] = {X -3.0337, Y 11.5717, Z -8.0000, A 0.000, B 0.000, C 0.000 }
gfCNCPoint6[3195] = {X -2.4098, Y 10.8371, Z -8.0000, A 0.000, B 0.000, C 0.000 }
gfCNCPoint6[3196] = {X -1.6337, Y 10.2658, Z -8.0000, A 0.000, B 0.000, C 0.000 }
gfCNCPoint6[3197] = {X -1.0364, Y 9.9250, Z -8.0000, A 0.000, B 0.000, C 0.000 }
gfCNCPoint6[3198] = {X -0.1704, Y 9.5539, Z -8.0000, A 0.000, B 0.000, C 0.000 }
gfCNCPoint6[3199] = {X 0.7568, Y 9.3871, Z -8.0000, A 0.000, B 0.000, C 0.000 }
gfCNCPoint6[3200] = {X 1.6978, Y 9.4332, Z -8.0000, A 0.000, B 0.000, C 0.000 }
gfCNCPoint6[3201] = {X 2.6043, Y 9.6899, Z -8.0000, A 0.000, B 0.000, C 0.000 }
gfCNCPoint6[3202] = {X 3.5530, Y 9.2656, Z -8.0000, A 0.000, B 0.000, C 0.000 }
gfCNCPoint6[3203] = {X 5.6159, Y 8.4884, Z -8.0000, A 0.000, B 0.000, C 0.000 }
gfCNCPoint6[3204] = {X 7.7422, Y 7.9067, Z -8.0000, A 0.000, B 0.000, C 0.000 }
gfCNCPoint6[3205] = {X 9.9135, Y 7.5257, Z -8.0000, A 0.000, B 0.000, C 0.000 }
gfCNCPoint6[3206] = {X 12.1108, Y 7.3486, Z -8.0000, A 0.000, B 0.000, C 0.000 }
gfCNCPoint6[3207] = {X 14.3150, Y 7.3769, Z -8.0000, A 0.000, B 0.000, C 0.000 }
gfCNCPoint6[3208] = {X 16.5071, Y 7.6104, Z -8.0000, A 0.000, B 0.000, C 0.000 }
gfCNCPoint6[3209] = {X 18.2268, Y 7.9616, Z -8.0000, A 0.000, B 0.000, C 0.000 }
gfCNCPoint6[3210] = {X 19.9019, Y 8.4858, Z -8.0000, A 0.000, B 0.000, C 0.000 }
gfCNCPoint6[3211] = {X 21.5151, Y 9.1776, Z -8.0000, A 0.000, B 0.000, C 0.000 }
gfCNCPoint6[3212] = {X 23.0495, Y 10.0298, Z -8.0000, A 0.000, B 0.000, C 0.000 }
gfCNCPoint6[3213] = {X 24.4894, Y 11.0336, Z -8.0000, A 0.000, B 0.000, C 0.000 }
gfCNCPoint6[3214] = {X 25.5614, Y 11.9710, Z -8.0000, A 0.000, B 0.000, C 0.000 }
gfCNCPoint6[3215] = {X 26.5231, Y 13.0213, Z -8.0000, A 0.000, B 0.000, C 0.000 }
gfCNCPoint6[3216] = {X 27.3626, Y 14.1716, Z -8.0000, A 0.000, B 0.000, C 0.000 }
gfCNCPoint6[3217] = {X 28.0696, Y 15.4078, Z -8.0000, A 0.000, B 0.000, C 0.000 }
gfCNCPoint6[3218] = {X 28.6354, Y 16.7147, Z -8.0000, A 0.000, B 0.000, C 0.000 }
gfCNCPoint6[3219] = {X 29.1046, Y 18.3531, Z -8.0000, A 0.000, B 0.000, C 0.000 }
gfCNCPoint6[3220] = {X 29.3830, Y 20.0344, Z -8.0000, A 0.000, B 0.000, C 0.000 }
gfCNCPoint6[3221] = {X 29.4669, Y 21.7366, Z -8.0000, A 0.000, B 0.000, C 0.000 }
gfCNCPoint6[3222] = {X 29.3552, Y 23.4372, Z -8.0000, A 0.000, B 0.000, C 0.000 }
gfCNCPoint6[3223] = {X 29.0494, Y 25.1138, Z -8.0000, A 0.000, B 0.000, C 0.000 }
gfCNCPoint6[3224] = {X 28.5906, Y 26.5986, Z -8.0000, A 0.000, B 0.000, C 0.000 }
gfCNCPoint6[3225] = {X 27.9365, Y 28.0082, Z -8.0000, A 0.000, B 0.000, C 0.000 }
gfCNCPoint6[3226] = {X 27.0989, Y 29.3171, Z -8.0000, A 0.000, B 0.000, C 0.000 }
gfCNCPoint6[3227] = {X 26.0930, Y 30.5016, Z -8.0000, A 0.000, B 0.000, C 0.000 }
gfCNCPoint6[3228] = {X 24.9370, Y 31.5402, Z -8.0000, A 0.000, B 0.000, C 0.000 }
gfCNCPoint6[3229] = {X 25.1525, Y 31.5961, Z -8.0000, A 0.000, B 0.000, C 0.000 }
gfCNCPoint6[3230] = {X 25.3647, Y 31.6635, Z -8.0000, A 0.000, B 0.000, C 0.000 }
gfCNCPoint6[3231] = {X 26.0979, Y 32.0010, Z -8.0000, A 0.000, B 0.000, C 0.000 }
gfCNCPoint6[3232] = {X 26.7522, Y 32.4736, Z -8.0000, A 0.000, B 0.000, C 0.000 }
gfCNCPoint6[3233] = {X 27.3028, Y 33.0637, Z -8.0000, A 0.000, B 0.000, C 0.000 }
gfCNCPoint6[3234] = {X 27.7292, Y 33.7491, Z -8.0000, A 0.000, B 0.000, C 0.000 }
gfCNCPoint6[3235] = {X 30.7660, Y 40.0227, Z -8.0000, A 0.000, B 0.000, C 0.000 }
gfCNCPoint6[3236] = {X 31.0747, Y 40.8982, Z -8.0000, A 0.000, B 0.000, C 0.000 }
gfCNCPoint6[3237] = {X 31.1815, Y 41.8203, Z -8.0000, A 0.000, B 0.000, C 0.000 }
gfCNCPoint6[3238] = {X 31.0813, Y 42.7431, Z -8.0000, A 0.000, B 0.000, C 0.000 }
gfCNCPoint6[3239] = {X 30.7789, Y 43.6208, Z -8.0000, A 0.000, B 0.000, C 0.000 }
gfCNCPoint6[3240] = {X 30.2893, Y 44.4095, Z -8.0000, A 0.000, B 0.000, C 0.000 }
gfCNCPoint6[3241] = {X 29.6371, Y 45.0700, Z -8.0000, A 0.000, B 0.000, C 0.000 }
gfCNCPoint6[3242] = {X 29.1011, Y 45.5034, Z -8.0000, A 0.000, B 0.000, C 0.000 }
gfCNCPoint6[3243] = {X 28.4113, Y 45.9566, Z -8.0000, A 0.000, B 0.000, C 0.000 }
gfCNCPoint6[3244] = {X 27.6458, Y 46.2650, Z -8.0000, A 0.000, B 0.000, C 0.000 }
gfCNCPoint6[3245] = {X 26.8345, Y 46.4166, Z -8.0000, A 0.000, B 0.000, C 0.000 }
gfCNCPoint6[3246] = {X 26.0092, Y 46.4054, Z -8.0000, A 0.000, B 0.000, C 0.000 }
gfCNCPoint6[3247] = {X 25.2024, Y 46.2318, Z -8.0000, A 0.000, B 0.000, C 0.000 }
gfCNCPoint6[3248] = {X 23.3927, Y 47.1902, Z -8.0000, A 0.000, B 0.000, C 0.000 }
gfCNCPoint6[3249] = {X 21.5205, Y 48.0197, Z -8.0000, A 0.000, B 0.000, C 0.000 }
gfCNCPoint6[3250] = {X 19.5948, Y 48.7162, Z -8.0000, A 0.000, B 0.000, C 0.000 }
gfCNCPoint6[3251] = {X 17.6684, Y 49.2602, Z -8.0000, A 0.000, B 0.000, C 0.000 }
gfCNCPoint6[3252] = {X 15.7013, Y 49.6315, Z -8.0000, A 0.000, B 0.000, C 0.000 }
gfCNCPoint6[3253] = {X 13.7091, Y 49.8272, Z -8.0000, A 0.000, B 0.000, C 0.000 }
gfCNCPoint6[3254] = {X 11.7074, Y 49.8458, Z -8.0000, A 0.000, B 0.000, C 0.000 }
gfCNCPoint6[3255] = {X 9.7119, Y 49.6872, Z -8.0000, A 0.000, B 0.000, C 0.000 }
gfCNCPoint6[3256] = {X 7.7383, Y 49.3525, Z -8.0000, A 0.000, B 0.000, C 0.000 }
gfCNCPoint6[3257] = {X 5.8547, Y 48.8365, Z -8.0000, A 0.000, B 0.000, C 0.000 }
gfCNCPoint6[3258] = {X 4.0450, Y 48.1023, Z -8.0000, A 0.000, B 0.000, C 0.000 }
gfCNCPoint6[3259] = {X 2.3343, Y 47.1600, Z -8.0000, A 0.000, B 0.000, C 0.000 }
gfCNCPoint6[3260] = {X 0.7466, Y 46.0228, Z -8.0000, A 0.000, B 0.000, C 0.000 }
gfCNCPoint6[3261] = {X -0.3714, Y 45.0175, Z -8.0000, A 0.000, B 0.000, C 0.000 }
gfCNCPoint6[3262] = {X -1.3646, Y 43.8886, Z -8.0000, A 0.000, B 0.000, C 0.000 }
gfCNCPoint6[3263] = {X -2.2192, Y 42.6515, Z -8.0000, A 0.000, B 0.000, C 0.000 }
gfCNCPoint6[3264] = {X -2.9236, Y 41.3232, Z -8.0000, A 0.000, B 0.000, C 0.000 }
gfCNCPoint6[3265] = {X -3.4683, Y 39.9218, Z -8.0000, A 0.000, B 0.000, C 0.000 }
gfCNCPoint6[3266] = {X -3.5889, Y 39.5266, Z -8.0000, A 0.000, B 0.000, C 0.000 }
gfCNCPoint6[3267] = {X -3.6967, Y 39.1278, Z -8.0000, A 0.000, B 0.000, C 0.000 }
gfCNCPoint6[3268] = {X -4.6784, Y 35.2501, Z -8.0000, A 0.000, B 0.000, C 0.000 }
gfCNCPoint6[3269] = {X -8.0070, Y 35.2296, Z -8.0000, A 0.000, B 0.000, C 0.000 }
gfCNCPoint6[3270] = {X -8.0070, Y 35.2296, Z -5.0000, A 0.000, B 0.000, C 0.000 }
gfCNCPoint6[3271] = {X -8.0070, Y 35.2296, Z 11.0000, A 0.000, B 0.000, C 0.000 }
gfCNCPoint6[3272] = {X -7.9995, Y 34.8051, Z 11.0000, A 0.000, B 0.000, C 0.000 }
gfCNCPoint6[3273] = {X -7.9995, Y 34.8051, Z -5.0000, A 0.000, B 0.000, C 0.000 }
gfCNCPoint6[3274] = {X -7.9995, Y 34.8051, Z -8.0000, A 0.000, B 0.000, C 0.000 }
gfCNCPoint6[3275] = {X -4.8514, Y 34.8967, Z -8.0000, A 0.000, B 0.000, C 0.000 }
gfCNCPoint6[3276] = {X -3.6967, Y 31.0670, Z -8.0000, A 0.000, B 0.000, C 0.000 }
gfCNCPoint6[3277] = {X -3.6591, Y 30.9444, Z -8.0000, A 0.000, B 0.000, C 0.000 }
gfCNCPoint6[3278] = {X -3.6205, Y 30.8221, Z -8.0000, A 0.000, B 0.000, C 0.000 }
gfCNCPoint6[3279] = {X -3.4463, Y 30.3106, Z -8.0000, A 0.000, B 0.000, C 0.000 }
gfCNCPoint6[3280] = {X -3.2535, Y 29.8059, Z -8.0000, A 0.000, B 0.000, C 0.000 }
gfCNCPoint6[3281] = {X -2.6189, Y 28.4661, Z -8.0000, A 0.000, B 0.000, C 0.000 }
gfCNCPoint6[3282] = {X -1.8072, Y 27.2256, Z -8.0000, A 0.000, B 0.000, C 0.000 }
gfCNCPoint6[3283] = {X -0.8336, Y 26.1075, Z -8.0000, A 0.000, B 0.000, C 0.000 }
gfCNCPoint6[3284] = {X 0.2836, Y 25.1329, Z -8.0000, A 0.000, B 0.000, C 0.000 }
gfCNCPoint6[3285] = {X 1.5234, Y 24.3201, Z -8.0000, A 0.000, B 0.000, C 0.000 }
gfCNCPoint6[3286] = {X 0.7353, Y 23.9292, Z -8.0000, A 0.000, B 0.000, C 0.000 }
gfCNCPoint6[3287] = {X 0.0428, Y 23.3868, Z -8.0000, A 0.000, B 0.000, C 0.000 }
gfCNCPoint6[3288] = {X -0.5255, Y 22.7153, Z -8.0000, A 0.000, B 0.000, C 0.000 }
gfCNCPoint6[3289] = {X -0.9460, Y 21.9427, Z -8.0000, A 0.000, B 0.000, C 0.000 }
gfCNCPoint6[3290] = {X -3.6217, Y 15.3838, Z -8.0000, A 0.000, B 0.000, C 0.000 }
gfCNCPoint6[3291] = {X -3.6607, Y 15.2744, Z -8.0000, A 0.000, B 0.000, C 0.000 }
gfCNCPoint6[3292] = {X -3.6967, Y 15.1641, Z -8.0000, A 0.000, B 0.000, C 0.000 }
gfCNCPoint6[3293] = {X -4.8865, Y 11.3451, Z -8.0000, A 0.000, B 0.000, C 0.000 }
gfCNCPoint6[3294] = {X -7.6967, Y 11.3451, Z -8.0000, A 0.000, B 0.000, C 0.000 }
gfCNCPoint6[3295] = {X -7.6967, Y 11.3451, Z -5.0000, A 0.000, B 0.000, C 0.000 }
gfCNCPoint6[3296] = {X -7.6967, Y 11.3451, Z 11.0000, A 0.000, B 0.000, C 0.000 }
gfCNCPoint6[3297] = {X -8.0066, Y 35.1739, Z 11.0000, A 0.000, B 0.000, C 0.000 }
gfCNCPoint6[3298] = {X -8.0066, Y 35.1739, Z -5.0000, A 0.000, B 0.000, C 0.000 }
gfCNCPoint6[3299] = {X -8.0066, Y 35.1739, Z -8.0000, A 0.000, B 0.000, C 0.000 }
gfCNCPoint6[3300] = {X -4.7800, Y 35.2035, Z -8.0000, A 0.000, B 0.000, C 0.000 }
gfCNCPoint6[3301] = {X -3.6967, Y 31.3530, Z -8.0000, A 0.000, B 0.000, C 0.000 }
gfCNCPoint6[3302] = {X -3.6228, Y 31.0990, Z -8.0000, A 0.000, B 0.000, C 0.000 }
gfCNCPoint6[3303] = {X -3.5443, Y 30.8465, Z -8.0000, A 0.000, B 0.000, C 0.000 }
gfCNCPoint6[3304] = {X -3.3710, Y 30.3377, Z -8.0000, A 0.000, B 0.000, C 0.000 }
gfCNCPoint6[3305] = {X -3.1791, Y 29.8355, Z -8.0000, A 0.000, B 0.000, C 0.000 }
gfCNCPoint6[3306] = {X -2.5652, Y 28.5342, Z -8.0000, A 0.000, B 0.000, C 0.000 }
gfCNCPoint6[3307] = {X -1.7830, Y 27.3266, Z -8.0000, A 0.000, B 0.000, C 0.000 }
gfCNCPoint6[3308] = {X -0.8465, Y 26.2343, Z -8.0000, A 0.000, B 0.000, C 0.000 }
gfCNCPoint6[3309] = {X 0.2275, Y 25.2768, Z -8.0000, A 0.000, B 0.000, C 0.000 }
gfCNCPoint6[3310] = {X 1.4198, Y 24.4715, Z -8.0000, A 0.000, B 0.000, C 0.000 }
gfCNCPoint6[3311] = {X 1.5686, Y 24.3865, Z -8.0000, A 0.000, B 0.000, C 0.000 }
gfCNCPoint6[3312] = {X 1.7186, Y 24.3039, Z -8.0000, A 0.000, B 0.000, C 0.000 }
gfCNCPoint6[3313] = {X 0.8915, Y 23.9306, Z -8.0000, A 0.000, B 0.000, C 0.000 }
gfCNCPoint6[3314] = {X 0.1628, Y 23.3899, Z -8.0000, A 0.000, B 0.000, C 0.000 }
gfCNCPoint6[3315] = {X -0.4343, Y 22.7066, Z -8.0000, A 0.000, B 0.000, C 0.000 }
gfCNCPoint6[3316] = {X -0.8722, Y 21.9118, Z -8.0000, A 0.000, B 0.000, C 0.000 }
gfCNCPoint6[3317] = {X -3.5467, Y 15.3559, Z -8.0000, A 0.000, B 0.000, C 0.000 }
gfCNCPoint6[3318] = {X -3.6292, Y 15.1113, Z -8.0000, A 0.000, B 0.000, C 0.000 }
gfCNCPoint6[3319] = {X -3.6967, Y 14.8621, Z -8.0000, A 0.000, B 0.000, C 0.000 }
gfCNCPoint6[3320] = {X -4.6241, Y 10.9711, Z -8.0000, A 0.000, B 0.000, C 0.000 }
gfCNCPoint6[3321] = {X -7.6967, Y 10.9711, Z -8.0000, A 0.000, B 0.000, C 0.000 }
gfCNCPoint6[3322] = {X -7.6967, Y 10.9711, Z -5.0000, A 0.000, B 0.000, C 0.000 }
gfCNCPoint6[3323] = {X -7.6967, Y 10.9711, Z 11.0000, A 0.000, B 0.000, C 0.000 }
gfCNCPoint6[3324] = {X -8.0059, Y 35.5717, Z 11.0000, A 0.000, B 0.000, C 0.000 }
gfCNCPoint6[3325] = {X -8.0059, Y 35.5717, Z -5.0000, A 0.000, B 0.000, C 0.000 }
gfCNCPoint6[3326] = {X -8.0059, Y 35.5717, Z -8.0000, A 0.000, B 0.000, C 0.000 }
gfCNCPoint6[3327] = {X -4.7023, Y 35.5309, Z -8.0000, A 0.000, B 0.000, C 0.000 }
gfCNCPoint6[3328] = {X -3.6967, Y 31.6593, Z -8.0000, A 0.000, B 0.000, C 0.000 }
gfCNCPoint6[3329] = {X -3.5879, Y 31.2635, Z -8.0000, A 0.000, B 0.000, C 0.000 }
gfCNCPoint6[3330] = {X -3.4681, Y 30.8709, Z -8.0000, A 0.000, B 0.000, C 0.000 }
gfCNCPoint6[3331] = {X -3.2956, Y 30.3647, Z -8.0000, A 0.000, B 0.000, C 0.000 }
gfCNCPoint6[3332] = {X -3.1048, Y 29.8651, Z -8.0000, A 0.000, B 0.000, C 0.000 }
gfCNCPoint6[3333] = {X -2.4955, Y 28.5734, Z -8.0000, A 0.000, B 0.000, C 0.000 }
gfCNCPoint6[3334] = {X -1.7191, Y 27.3746, Z -8.0000, A 0.000, B 0.000, C 0.000 }
gfCNCPoint6[3335] = {X -0.7895, Y 26.2904, Z -8.0000, A 0.000, B 0.000, C 0.000 }
gfCNCPoint6[3336] = {X 0.2766, Y 25.3400, Z -8.0000, A 0.000, B 0.000, C 0.000 }
gfCNCPoint6[3337] = {X 1.4601, Y 24.5406, Z -8.0000, A 0.000, B 0.000, C 0.000 }
gfCNCPoint6[3338] = {X 1.6925, Y 24.4092, Z -8.0000, A 0.000, B 0.000, C 0.000 }
gfCNCPoint6[3339] = {X 1.9281, Y 24.2837, Z -8.0000, A 0.000, B 0.000, C 0.000 }
gfCNCPoint6[3340] = {X 1.0580, Y 23.9327, Z -8.0000, A 0.000, B 0.000, C 0.000 }
gfCNCPoint6[3341] = {X 0.2886, Y 23.3958, Z -8.0000, A 0.000, B 0.000, C 0.000 }
gfCNCPoint6[3342] = {X -0.3408, Y 22.7000, Z -8.0000, A 0.000, B 0.000, C 0.000 }
gfCNCPoint6[3343] = {X -0.7984, Y 21.8809, Z -8.0000, A 0.000, B 0.000, C 0.000 }
gfCNCPoint6[3344] = {X -3.4717, Y 15.3281, Z -8.0000, A 0.000, B 0.000, C 0.000 }
gfCNCPoint6[3345] = {X -3.6097, Y 14.8812, Z -8.0000, A 0.000, B 0.000, C 0.000 }
gfCNCPoint6[3346] = {X -3.6967, Y 14.4216, Z -8.0000, A 0.000, B 0.000, C 0.000 }
gfCNCPoint6[3347] = {X -4.2183, Y 10.4558, Z -8.0000, A 0.000, B 0.000, C 0.000 }
gfCNCPoint6[3348] = {X -7.6967, Y 10.4558, Z -8.0000, A 0.000, B 0.000, C 0.000 }
gfCNCPoint6[3349] = {X -7.6967, Y 10.4558, Z -5.0000, A 0.000, B 0.000, C 0.000 }
gfCNCPoint6[3350] = {X -7.6967, Y 10.4558, Z 11.0000, A 0.000, B 0.000, C 0.000 }
gfCNCPoint6[3351] = {X -7.9955, Y 36.0055, Z 11.0000, A 0.000, B 0.000, C 0.000 }
gfCNCPoint6[3352] = {X -7.9955, Y 36.0055, Z -5.0000, A 0.000, B 0.000, C 0.000 }
gfCNCPoint6[3353] = {X -7.9955, Y 36.0055, Z -8.0000, A 0.000, B 0.000, C 0.000 }
gfCNCPoint6[3354] = {X -4.6166, Y 35.8844, Z -8.0000, A 0.000, B 0.000, C 0.000 }
gfCNCPoint6[3355] = {X -3.6967, Y 31.9917, Z -8.0000, A 0.000, B 0.000, C 0.000 }
gfCNCPoint6[3356] = {X -3.5550, Y 31.4405, Z -8.0000, A 0.000, B 0.000, C 0.000 }
gfCNCPoint6[3357] = {X -3.3920, Y 30.8953, Z -8.0000, A 0.000, B 0.000, C 0.000 }
gfCNCPoint6[3358] = {X -3.2203, Y 30.3916, Z -8.0000, A 0.000, B 0.000, C 0.000 }
gfCNCPoint6[3359] = {X -3.0304, Y 29.8946, Z -8.0000, A 0.000, B 0.000, C 0.000 }
gfCNCPoint6[3360] = {X -2.4257, Y 28.6125, Z -8.0000, A 0.000, B 0.000, C 0.000 }
gfCNCPoint6[3361] = {X -1.6551, Y 27.4227, Z -8.0000, A 0.000, B 0.000, C 0.000 }
gfCNCPoint6[3362] = {X -0.7325, Y 26.3465, Z -8.0000, A 0.000, B 0.000, C 0.000 }
gfCNCPoint6[3363] = {X 0.3256, Y 25.4032, Z -8.0000, A 0.000, B 0.000, C 0.000 }
gfCNCPoint6[3364] = {X 1.5003, Y 24.6097, Z -8.0000, A 0.000, B 0.000, C 0.000 }
gfCNCPoint6[3365] = {X 1.8253, Y 24.4282, Z -8.0000, A 0.000, B 0.000, C 0.000 }
gfCNCPoint6[3366] = {X 2.1565, Y 24.2581, Z -8.0000, A 0.000, B 0.000, C 0.000 }
gfCNCPoint6[3367] = {X 1.2382, Y 23.9358, Z -8.0000, A 0.000, B 0.000, C 0.000 }
gfCNCPoint6[3368] = {X 0.4225, Y 23.4052, Z -8.0000, A 0.000, B 0.000, C 0.000 }
gfCNCPoint6[3369] = {X -0.2445, Y 22.6965, Z -8.0000, A 0.000, B 0.000, C 0.000 }
gfCNCPoint6[3370] = {X -0.7246, Y 21.8500, Z -8.0000, A 0.000, B 0.000, C 0.000 }
gfCNCPoint6[3371] = {X -3.3967, Y 15.3002, Z -8.0000, A 0.000, B 0.000, C 0.000 }
gfCNCPoint6[3372] = {X -3.6236, Y 14.3618, Z -8.0000, A 0.000, B 0.000, C 0.000 }
gfCNCPoint6[3373] = {X -3.6236, Y 13.3964, Z -8.0000, A 0.000, B 0.000, C 0.000 }
gfCNCPoint6[3374] = {X -3.3967, Y 12.4580, Z -8.0000, A 0.000, B 0.000, C 0.000 }
gfCNCPoint6[3375] = {X -2.9671, Y 11.6161, Z -8.0000, A 0.000, B 0.000, C 0.000 }
gfCNCPoint6[3376] = {X -2.3552, Y 10.8956, Z -8.0000, A 0.000, B 0.000, C 0.000 }
gfCNCPoint6[3377] = {X -1.5940, Y 10.3353, Z -8.0000, A 0.000, B 0.000, C 0.000 }
gfCNCPoint6[3378] = {X -0.9967, Y 9.9945, Z -8.0000, A 0.000, B 0.000, C 0.000 }
gfCNCPoint6[3379] = {X -0.1386, Y 9.6279, Z -8.0000, A 0.000, B 0.000, C 0.000 }
gfCNCPoint6[3380] = {X 0.7803, Y 9.4658, Z -8.0000, A 0.000, B 0.000, C 0.000 }
gfCNCPoint6[3381] = {X 1.7121, Y 9.5167, Z -8.0000, A 0.000, B 0.000, C 0.000 }
gfCNCPoint6[3382] = {X 2.6079, Y 9.7781, Z -8.0000, A 0.000, B 0.000, C 0.000 }
gfCNCPoint6[3383] = {X 3.5852, Y 9.3388, Z -8.0000, A 0.000, B 0.000, C 0.000 }
gfCNCPoint6[3384] = {X 5.6410, Y 8.5643, Z -8.0000, A 0.000, B 0.000, C 0.000 }
gfCNCPoint6[3385] = {X 7.7601, Y 7.9847, Z -8.0000, A 0.000, B 0.000, C 0.000 }
gfCNCPoint6[3386] = {X 9.9239, Y 7.6050, Z -8.0000, A 0.000, B 0.000, C 0.000 }
gfCNCPoint6[3387] = {X 12.1137, Y 7.4285, Z -8.0000, A 0.000, B 0.000, C 0.000 }
gfCNCPoint6[3388] = {X 14.3104, Y 7.4567, Z -8.0000, A 0.000, B 0.000, C 0.000 }
gfCNCPoint6[3389] = {X 16.4949, Y 7.6895, Z -8.0000, A 0.000, B 0.000, C 0.000 }
gfCNCPoint6[3390] = {X 18.2067, Y 8.0391, Z -8.0000, A 0.000, B 0.000, C 0.000 }
gfCNCPoint6[3391] = {X 19.8741, Y 8.5608, Z -8.0000, A 0.000, B 0.000, C 0.000 }
gfCNCPoint6[3392] = {X 21.4798, Y 9.2494, Z -8.0000, A 0.000, B 0.000, C 0.000 }
gfCNCPoint6[3393] = {X 23.0072, Y 10.0977, Z -8.0000, A 0.000, B 0.000, C 0.000 }
gfCNCPoint6[3394] = {X 24.4404, Y 11.0968, Z -8.0000, A 0.000, B 0.000, C 0.000 }
gfCNCPoint6[3395] = {X 25.5056, Y 12.0283, Z -8.0000, A 0.000, B 0.000, C 0.000 }
gfCNCPoint6[3396] = {X 26.4611, Y 13.0719, Z -8.0000, A 0.000, B 0.000, C 0.000 }
gfCNCPoint6[3397] = {X 27.2953, Y 14.2149, Z -8.0000, A 0.000, B 0.000, C 0.000 }
gfCNCPoint6[3398] = {X 27.9978, Y 15.4432, Z -8.0000, A 0.000, B 0.000, C 0.000 }
gfCNCPoint6[3399] = {X 28.5601, Y 16.7417, Z -8.0000, A 0.000, B 0.000, C 0.000 }
gfCNCPoint6[3400] = {X 29.0267, Y 18.3712, Z -8.0000, A 0.000, B 0.000, C 0.000 }
gfCNCPoint6[3401] = {X 29.3035, Y 20.0434, Z -8.0000, A 0.000, B 0.000, C 0.000 }
gfCNCPoint6[3402] = {X 29.3869, Y 21.7364, Z -8.0000, A 0.000, B 0.000, C 0.000 }
gfCNCPoint6[3403] = {X 29.2758, Y 23.4277, Z -8.0000, A 0.000, B 0.000, C 0.000 }
gfCNCPoint6[3404] = {X 28.9716, Y 25.0952, Z -8.0000, A 0.000, B 0.000, C 0.000 }
gfCNCPoint6[3405] = {X 28.5035, Y 26.6020, Z -8.0000, A 0.000, B 0.000, C 0.000 }
gfCNCPoint6[3406] = {X 27.8329, Y 28.0302, Z -8.0000, A 0.000, B 0.000, C 0.000 }
gfCNCPoint6[3407] = {X 26.9725, Y 29.3527, Z -8.0000, A 0.000, B 0.000, C 0.000 }
gfCNCPoint6[3408] = {X 25.9385, Y 30.5445, Z -8.0000, A 0.000, B 0.000, C 0.000 }
gfCNCPoint6[3409] = {X 24.7506, Y 31.5830, Z -8.0000, A 0.000, B 0.000, C 0.000 }
gfCNCPoint6[3410] = {X 25.0475, Y 31.6501, Z -8.0000, A 0.000, B 0.000, C 0.000 }
gfCNCPoint6[3411] = {X 25.3385, Y 31.7391, Z -8.0000, A 0.000, B 0.000, C 0.000 }
gfCNCPoint6[3412] = {X 26.0576, Y 32.0700, Z -8.0000, A 0.000, B 0.000, C 0.000 }
gfCNCPoint6[3413] = {X 26.6993, Y 32.5336, Z -8.0000, A 0.000, B 0.000, C 0.000 }
gfCNCPoint6[3414] = {X 27.2393, Y 33.1124, Z -8.0000, A 0.000, B 0.000, C 0.000 }
gfCNCPoint6[3415] = {X 27.6575, Y 33.7845, Z -8.0000, A 0.000, B 0.000, C 0.000 }
gfCNCPoint6[3416] = {X 30.6940, Y 40.0576, Z -8.0000, A 0.000, B 0.000, C 0.000 }
gfCNCPoint6[3417] = {X 30.9967, Y 40.9162, Z -8.0000, A 0.000, B 0.000, C 0.000 }
gfCNCPoint6[3418] = {X 31.1015, Y 41.8206, Z -8.0000, A 0.000, B 0.000, C 0.000 }
gfCNCPoint6[3419] = {X 31.0032, Y 42.7257, Z -8.0000, A 0.000, B 0.000, C 0.000 }
gfCNCPoint6[3420] = {X 30.7066, Y 43.5864, Z -8.0000, A 0.000, B 0.000, C 0.000 }
gfCNCPoint6[3421] = {X 30.2265, Y 44.3600, Z -8.0000, A 0.000, B 0.000, C 0.000 }
gfCNCPoint6[3422] = {X 29.5868, Y 45.0078, Z -8.0000, A 0.000, B 0.000, C 0.000 }
gfCNCPoint6[3423] = {X 29.0508, Y 45.4413, Z -8.0000, A 0.000, B 0.000, C 0.000 }
gfCNCPoint6[3424] = {X 28.3680, Y 45.8890, Z -8.0000, A 0.000, B 0.000, C 0.000 }
gfCNCPoint6[3425] = {X 27.6098, Y 46.1921, Z -8.0000, A 0.000, B 0.000, C 0.000 }
gfCNCPoint6[3426] = {X 26.8065, Y 46.3386, Z -8.0000, A 0.000, B 0.000, C 0.000 }
gfCNCPoint6[3427] = {X 25.9902, Y 46.3226, Z -8.0000, A 0.000, B 0.000, C 0.000 }
gfCNCPoint6[3428] = {X 25.1933, Y 46.1447, Z -8.0000, A 0.000, B 0.000, C 0.000 }
gfCNCPoint6[3429] = {X 23.3790, Y 47.1079, Z -8.0000, A 0.000, B 0.000, C 0.000 }
gfCNCPoint6[3430] = {X 21.5015, Y 47.9411, Z -8.0000, A 0.000, B 0.000, C 0.000 }
gfCNCPoint6[3431] = {X 19.5700, Y 48.6402, Z -8.0000, A 0.000, B 0.000, C 0.000 }
gfCNCPoint6[3432] = {X 17.6503, Y 49.1822, Z -8.0000, A 0.000, B 0.000, C 0.000 }
gfCNCPoint6[3433] = {X 15.6901, Y 49.5523, Z -8.0000, A 0.000, B 0.000, C 0.000 }
gfCNCPoint6[3434] = {X 13.7049, Y 49.7473, Z -8.0000, A 0.000, B 0.000, C 0.000 }
gfCNCPoint6[3435] = {X 11.7102, Y 49.7659, Z -8.0000, A 0.000, B 0.000, C 0.000 }
gfCNCPoint6[3436] = {X 9.7217, Y 49.6078, Z -8.0000, A 0.000, B 0.000, C 0.000 }
gfCNCPoint6[3437] = {X 7.7550, Y 49.2743, Z -8.0000, A 0.000, B 0.000, C 0.000 }
gfCNCPoint6[3438] = {X 5.8804, Y 48.7608, Z -8.0000, A 0.000, B 0.000, C 0.000 }
gfCNCPoint6[3439] = {X 4.0794, Y 48.0301, Z -8.0000, A 0.000, B 0.000, C 0.000 }
gfCNCPoint6[3440] = {X 2.3769, Y 47.0923, Z -8.0000, A 0.000, B 0.000, C 0.000 }
gfCNCPoint6[3441] = {X 0.7968, Y 45.9605, Z -8.0000, A 0.000, B 0.000, C 0.000 }
gfCNCPoint6[3442] = {X -0.3144, Y 44.9614, Z -8.0000, A 0.000, B 0.000, C 0.000 }
gfCNCPoint6[3443] = {X -1.3014, Y 43.8395, Z -8.0000, A 0.000, B 0.000, C 0.000 }
gfCNCPoint6[3444] = {X -2.1508, Y 42.6101, Z -8.0000, A 0.000, B 0.000, C 0.000 }
gfCNCPoint6[3445] = {X -2.8509, Y 41.2900, Z -8.0000, A 0.000, B 0.000, C 0.000 }
gfCNCPoint6[3446] = {X -3.3922, Y 39.8972, Z -8.0000, A 0.000, B 0.000, C 0.000 }
gfCNCPoint6[3447] = {X -3.5570, Y 39.3441, Z -8.0000, A 0.000, B 0.000, C 0.000 }
gfCNCPoint6[3448] = {X -3.6967, Y 38.7841, Z -8.0000, A 0.000, B 0.000, C 0.000 }
gfCNCPoint6[3449] = {X -4.5771, Y 34.8822, Z -8.0000, A 0.000, B 0.000, C 0.000 }
gfCNCPoint6[3450] = {X -7.9987, Y 34.7775, Z -8.0000, A 0.000, B 0.000, C 0.000 }
gfCNCPoint6[3451] = {X -7.9987, Y 34.7775, Z -5.0000, A 0.000, B 0.000, C 0.000 }
gfCNCPoint6[3452] = {X -7.9987, Y 34.7775, Z 11.0000, A 0.000, B 0.000, C 0.000 }
gfCNCPoint6[3453] = {X -7.9719, Y 36.4867, Z 11.0000, A 0.000, B 0.000, C 0.000 }
gfCNCPoint6[3454] = {X -7.9719, Y 36.4867, Z -5.0000, A 0.000, B 0.000, C 0.000 }
gfCNCPoint6[3455] = {X -7.9719, Y 36.4867, Z -8.0000, A 0.000, B 0.000, C 0.000 }
gfCNCPoint6[3456] = {X -4.5204, Y 36.2729, Z -8.0000, A 0.000, B 0.000, C 0.000 }
gfCNCPoint6[3457] = {X -3.6967, Y 32.3587, Z -8.0000, A 0.000, B 0.000, C 0.000 }
gfCNCPoint6[3458] = {X -3.5247, Y 31.6343, Z -8.0000, A 0.000, B 0.000, C 0.000 }
gfCNCPoint6[3459] = {X -3.3158, Y 30.9197, Z -8.0000, A 0.000, B 0.000, C 0.000 }
gfCNCPoint6[3460] = {X -3.1448, Y 30.4180, Z -8.0000, A 0.000, B 0.000, C 0.000 }
gfCNCPoint6[3461] = {X -2.9556, Y 29.9228, Z -8.0000, A 0.000, B 0.000, C 0.000 }
gfCNCPoint6[3462] = {X -2.3554, Y 28.6506, Z -8.0000, A 0.000, B 0.000, C 0.000 }
gfCNCPoint6[3463] = {X -1.5906, Y 27.4701, Z -8.0000, A 0.000, B 0.000, C 0.000 }
gfCNCPoint6[3464] = {X -0.6751, Y 26.4022, Z -8.0000, A 0.000, B 0.000, C 0.000 }
gfCNCPoint6[3465] = {X 0.3749, Y 25.4662, Z -8.0000, A 0.000, B 0.000, C 0.000 }
gfCNCPoint6[3466] = {X 1.5406, Y 24.6789, Z -8.0000, A 0.000, B 0.000, C 0.000 }
gfCNCPoint6[3467] = {X 1.9706, Y 24.4419, Z -8.0000, A 0.000, B 0.000, C 0.000 }
gfCNCPoint6[3468] = {X 2.4113, Y 24.2252, Z -8.0000, A 0.000, B 0.000, C 0.000 }
gfCNCPoint6[3469] = {X 1.6198, Y 24.0145, Z -8.0000, A 0.000, B 0.000, C 0.000 }
gfCNCPoint6[3470] = {X 0.8879, Y 23.6470, Z -8.0000, A 0.000, B 0.000, C 0.000 }
gfCNCPoint6[3471] = {X 0.2461, Y 23.1382, Z -8.0000, A 0.000, B 0.000, C 0.000 }
gfCNCPoint6[3472] = {X -0.2786, Y 22.5093, Z -8.0000, A 0.000, B 0.000, C 0.000 }
gfCNCPoint6[3473] = {X -0.6642, Y 21.7867, Z -8.0000, A 0.000, B 0.000, C 0.000 }
gfCNCPoint6[3474] = {X -3.2754, Y 15.3911, Z -8.0000, A 0.000, B 0.000, C 0.000 }
gfCNCPoint6[3475] = {X -3.2991, Y 15.3319, Z -8.0000, A 0.000, B 0.000, C 0.000 }
gfCNCPoint6[3476] = {X -3.3217, Y 15.2723, Z -8.0000, A 0.000, B 0.000, C 0.000 }
gfCNCPoint6[3477] = {X -3.5441, Y 14.3524, Z -8.0000, A 0.000, B 0.000, C 0.000 }
gfCNCPoint6[3478] = {X -3.5441, Y 13.4059, Z -8.0000, A 0.000, B 0.000, C 0.000 }
gfCNCPoint6[3479] = {X -3.3217, Y 12.4859, Z -8.0000, A 0.000, B 0.000, C 0.000 }
gfCNCPoint6[3480] = {X -2.9005, Y 11.6605, Z -8.0000, A 0.000, B 0.000, C 0.000 }
gfCNCPoint6[3481] = {X -2.3007, Y 10.9541, Z -8.0000, A 0.000, B 0.000, C 0.000 }
gfCNCPoint6[3482] = {X -1.5544, Y 10.4048, Z -8.0000, A 0.000, B 0.000, C 0.000 }
gfCNCPoint6[3483] = {X -0.9063, Y 10.0355, Z -8.0000, A 0.000, B 0.000, C 0.000 }
gfCNCPoint6[3484] = {X -0.1052, Y 9.7014, Z -8.0000, A 0.000, B 0.000, C 0.000 }
gfCNCPoint6[3485] = {X 0.7490, Y 9.5480, Z -8.0000, A 0.000, B 0.000, C 0.000 }
gfCNCPoint6[3486] = {X 1.6162, Y 9.5824, Z -8.0000, A 0.000, B 0.000, C 0.000 }
gfCNCPoint6[3487] = {X 2.4556, Y 9.8031, Z -8.0000, A 0.000, B 0.000, C 0.000 }
gfCNCPoint6[3488] = {X 2.5431, Y 9.8378, Z -8.0000, A 0.000, B 0.000, C 0.000 }
gfCNCPoint6[3489] = {X 2.6297, Y 9.8745, Z -8.0000, A 0.000, B 0.000, C 0.000 }
gfCNCPoint6[3490] = {X 2.6555, Y 9.8423, Z -8.0000, A 0.000, B 0.000, C 0.000 }
gfCNCPoint6[3491] = {X 3.6169, Y 9.4123, Z -8.0000, A 0.000, B 0.000, C 0.000 }
gfCNCPoint6[3492] = {X 5.6658, Y 8.6404, Z -8.0000, A 0.000, B 0.000, C 0.000 }
gfCNCPoint6[3493] = {X 7.7777, Y 8.0628, Z -8.0000, A 0.000, B 0.000, C 0.000 }
gfCNCPoint6[3494] = {X 9.9343, Y 7.6843, Z -8.0000, A 0.000, B 0.000, C 0.000 }
gfCNCPoint6[3495] = {X 12.1167, Y 7.5085, Z -8.0000, A 0.000, B 0.000, C 0.000 }
gfCNCPoint6[3496] = {X 14.3060, Y 7.5366, Z -8.0000, A 0.000, B 0.000, C 0.000 }
gfCNCPoint6[3497] = {X 16.4832, Y 7.7686, Z -8.0000, A 0.000, B 0.000, C 0.000 }
gfCNCPoint6[3498] = {X 18.1869, Y 8.1166, Z -8.0000, A 0.000, B 0.000, C 0.000 }
gfCNCPoint6[3499] = {X 19.8465, Y 8.6359, Z -8.0000, A 0.000, B 0.000, C 0.000 }
gfCNCPoint6[3500] = {X 21.4446, Y 9.3213, Z -8.0000, A 0.000, B 0.000, C 0.000 }
gfCNCPoint6[3501] = {X 22.9649, Y 10.1656, Z -8.0000, A 0.000, B 0.000, C 0.000 }
gfCNCPoint6[3502] = {X 24.3914, Y 11.1600, Z -8.0000, A 0.000, B 0.000, C 0.000 }
gfCNCPoint6[3503] = {X 25.4497, Y 12.0855, Z -8.0000, A 0.000, B 0.000, C 0.000 }
gfCNCPoint6[3504] = {X 26.3991, Y 13.1225, Z -8.0000, A 0.000, B 0.000, C 0.000 }
gfCNCPoint6[3505] = {X 27.2280, Y 14.2582, Z -8.0000, A 0.000, B 0.000, C 0.000 }
gfCNCPoint6[3506] = {X 27.9261, Y 15.4786, Z -8.0000, A 0.000, B 0.000, C 0.000 }
gfCNCPoint6[3507] = {X 28.4848, Y 16.7687, Z -8.0000, A 0.000, B 0.000, C 0.000 }
gfCNCPoint6[3508] = {X 28.9488, Y 18.3896, Z -8.0000, A 0.000, B 0.000, C 0.000 }
gfCNCPoint6[3509] = {X 29.2241, Y 20.0529, Z -8.0000, A 0.000, B 0.000, C 0.000 }
gfCNCPoint6[3510] = {X 29.3069, Y 21.7368, Z -8.0000, A 0.000, B 0.000, C 0.000 }
gfCNCPoint6[3511] = {X 29.1962, Y 23.4191, Z -8.0000, A 0.000, B 0.000, C 0.000 }
gfCNCPoint6[3512] = {X 28.8935, Y 25.0776, Z -8.0000, A 0.000, B 0.000, C 0.000 }
gfCNCPoint6[3513] = {X 28.4150, Y 26.6087, Z -8.0000, A 0.000, B 0.000, C 0.000 }
gfCNCPoint6[3514] = {X 27.7260, Y 28.0573, Z -8.0000, A 0.000, B 0.000, C 0.000 }
gfCNCPoint6[3515] = {X 26.8401, Y 29.3945, Z -8.0000, A 0.000, B 0.000, C 0.000 }
gfCNCPoint6[3516] = {X 25.7750, Y 30.5939, Z -8.0000, A 0.000, B 0.000, C 0.000 }
gfCNCPoint6[3517] = {X 24.5517, Y 31.6316, Z -8.0000, A 0.000, B 0.000, C 0.000 }
gfCNCPoint6[3518] = {X 24.9365, Y 31.7045, Z -8.0000, A 0.000, B 0.000, C 0.000 }
gfCNCPoint6[3519] = {X 25.3123, Y 31.8147, Z -8.0000, A 0.000, B 0.000, C 0.000 }
gfCNCPoint6[3520] = {X 26.0247, Y 32.1434, Z -8.0000, A 0.000, B 0.000, C 0.000 }
gfCNCPoint6[3521] = {X 26.6592, Y 32.6050, Z -8.0000, A 0.000, B 0.000, C 0.000 }
gfCNCPoint6[3522] = {X 27.1914, Y 33.1815, Z -8.0000, A 0.000, B 0.000, C 0.000 }
gfCNCPoint6[3523] = {X 27.6008, Y 33.8508, Z -8.0000, A 0.000, B 0.000, C 0.000 }
gfCNCPoint6[3524] = {X 30.6220, Y 40.0925, Z -8.0000, A 0.000, B 0.000, C 0.000 }
gfCNCPoint6[3525] = {X 30.9188, Y 40.9342, Z -8.0000, A 0.000, B 0.000, C 0.000 }
gfCNCPoint6[3526] = {X 31.0215, Y 41.8209, Z -8.0000, A 0.000, B 0.000, C 0.000 }
gfCNCPoint6[3527] = {X 30.9251, Y 42.7082, Z -8.0000, A 0.000, B 0.000, C 0.000 }
gfCNCPoint6[3528] = {X 30.6343, Y 43.5521, Z -8.0000, A 0.000, B 0.000, C 0.000 }
gfCNCPoint6[3529] = {X 30.1637, Y 44.3105, Z -8.0000, A 0.000, B 0.000, C 0.000 }
gfCNCPoint6[3530] = {X 29.5365, Y 44.9456, Z -8.0000, A 0.000, B 0.000, C 0.000 }
gfCNCPoint6[3531] = {X 29.0005, Y 45.3790, Z -8.0000, A 0.000, B 0.000, C 0.000 }
gfCNCPoint6[3532] = {X 28.1809, Y 45.8923, Z -8.0000, A 0.000, B 0.000, C 0.000 }
gfCNCPoint6[3533] = {X 27.2623, Y 46.1944, Z -8.0000, A 0.000, B 0.000, C 0.000 }
gfCNCPoint6[3534] = {X 26.2981, Y 46.2678, Z -8.0000, A 0.000, B 0.000, C 0.000 }
gfCNCPoint6[3535] = {X 25.3444, Y 46.1082, Z -8.0000, A 0.000, B 0.000, C 0.000 }
gfCNCPoint6[3536] = {X 25.2642, Y 46.0836, Z -8.0000, A 0.000, B 0.000, C 0.000 }
gfCNCPoint6[3537] = {X 25.1845, Y 46.0574, Z -8.0000, A 0.000, B 0.000, C 0.000 }
gfCNCPoint6[3538] = {X 23.3652, Y 47.0257, Z -8.0000, A 0.000, B 0.000, C 0.000 }
gfCNCPoint6[3539] = {X 21.4818, Y 47.8628, Z -8.0000, A 0.000, B 0.000, C 0.000 }
gfCNCPoint6[3540] = {X 19.5440, Y 48.5645, Z -8.0000, A 0.000, B 0.000, C 0.000 }
gfCNCPoint6[3541] = {X 17.6311, Y 49.1046, Z -8.0000, A 0.000, B 0.000, C 0.000 }
gfCNCPoint6[3542] = {X 15.6779, Y 49.4732, Z -8.0000, A 0.000, B 0.000, C 0.000 }
gfCNCPoint6[3543] = {X 13.6997, Y 49.6675, Z -8.0000, A 0.000, B 0.000, C 0.000 }
gfCNCPoint6[3544] = {X 11.7121, Y 49.6859, Z -8.0000, A 0.000, B 0.000, C 0.000 }
gfCNCPoint6[3545] = {X 9.7307, Y 49.5283, Z -8.0000, A 0.000, B 0.000, C 0.000 }
gfCNCPoint6[3546] = {X 7.7710, Y 49.1959, Z -8.0000, A 0.000, B 0.000, C 0.000 }
gfCNCPoint6[3547] = {X 5.9053, Y 48.6847, Z -8.0000, A 0.000, B 0.000, C 0.000 }
gfCNCPoint6[3548] = {X 4.1128, Y 47.9574, Z -8.0000, A 0.000, B 0.000, C 0.000 }
gfCNCPoint6[3549] = {X 2.4185, Y 47.0239, Z -8.0000, A 0.000, B 0.000, C 0.000 }
gfCNCPoint6[3550] = {X 0.8459, Y 45.8974, Z -8.0000, A 0.000, B 0.000, C 0.000 }
gfCNCPoint6[3551] = {X -0.2581, Y 44.9046, Z -8.0000, A 0.000, B 0.000, C 0.000 }
gfCNCPoint6[3552] = {X -1.2387, Y 43.7898, Z -8.0000, A 0.000, B 0.000, C 0.000 }
gfCNCPoint6[3553] = {X -2.0826, Y 42.5682, Z -8.0000, A 0.000, B 0.000, C 0.000 }
gfCNCPoint6[3554] = {X -2.7782, Y 41.2565, Z -8.0000, A 0.000, B 0.000, C 0.000 }
gfCNCPoint6[3555] = {X -3.3160, Y 39.8726, Z -8.0000, A 0.000, B 0.000, C 0.000 }
gfCNCPoint6[3556] = {X -3.5286, Y 39.1395, Z -8.0000, A 0.000, B 0.000, C 0.000 }
gfCNCPoint6[3557] = {X -3.6967, Y 38.3948, Z -8.0000, A 0.000, B 0.000, C 0.000 }
gfCNCPoint6[3558] = {X -4.4600, Y 34.4684, Z -8.0000, A 0.000, B 0.000, C 0.000 }
gfCNCPoint6[3559] = {X -7.9757, Y 34.2626, Z -8.0000, A 0.000, B 0.000, C 0.000 }
gfCNCPoint6[3560] = {X -7.9757, Y 34.2626, Z -5.0000, A 0.000, B 0.000, C 0.000 }
gfCNCPoint6[3561] = {X -7.9757, Y 34.2626, Z 11.0000, A 0.000, B 0.000, C 0.000 }
gfCNCPoint6[3562] = {X 39.8241, Y 26.3831, Z 11.0000, A 0.000, B 0.000, C 0.000 }
gfCNCPoint6[3563] = {X 39.8241, Y 26.3831, Z -5.0000, A 0.000, B 0.000, C 0.000 }
gfCNCPoint6[3564] = {X 39.8241, Y 26.3831, Z -8.0000, A 0.000, B 0.000, C 0.000 }
gfCNCPoint6[3565] = {X 43.6474, Y 27.8074, Z -8.0000, A 0.000, B 0.000, C 0.000 }
gfCNCPoint6[3566] = {X 48.2901, Y 15.3446, Z -8.0000, A 0.000, B 0.000, C 0.000 }
gfCNCPoint6[3567] = {X 47.9079, Y 14.6186, Z -8.0000, A 0.000, B 0.000, C 0.000 }
gfCNCPoint6[3568] = {X 47.6697, Y 13.8334, Z -8.0000, A 0.000, B 0.000, C 0.000 }
gfCNCPoint6[3569] = {X 47.5844, Y 13.0173, Z -8.0000, A 0.000, B 0.000, C 0.000 }
gfCNCPoint6[3570] = {X 47.5842, Y 12.1868, Z -8.0000, A 0.000, B 0.000, C 0.000 }
gfCNCPoint6[3571] = {X 47.6925, Y 11.2255, Z -8.0000, A 0.000, B 0.000, C 0.000 }
gfCNCPoint6[3572] = {X 48.0120, Y 10.3125, Z -8.0000, A 0.000, B 0.000, C 0.000 }
gfCNCPoint6[3573] = {X 48.5267, Y 9.4933, Z -8.0000, A 0.000, B 0.000, C 0.000 }
gfCNCPoint6[3574] = {X 49.2107, Y 8.8093, Z -8.0000, A 0.000, B 0.000, C 0.000 }
gfCNCPoint6[3575] = {X 50.0298, Y 8.2946, Z -8.0000, A 0.000, B 0.000, C 0.000 }
gfCNCPoint6[3576] = {X 50.9429, Y 7.9751, Z -8.0000, A 0.000, B 0.000, C 0.000 }
gfCNCPoint6[3577] = {X 51.9042, Y 7.8668, Z -8.0000, A 0.000, B 0.000, C 0.000 }
gfCNCPoint6[3578] = {X 59.6221, Y 7.8668, Z -8.0000, A 0.000, B 0.000, C 0.000 }
gfCNCPoint6[3579] = {X 60.5834, Y 7.9751, Z -8.0000, A 0.000, B 0.000, C 0.000 }
gfCNCPoint6[3580] = {X 61.4965, Y 8.2946, Z -8.0000, A 0.000, B 0.000, C 0.000 }
gfCNCPoint6[3581] = {X 62.3156, Y 8.8093, Z -8.0000, A 0.000, B 0.000, C 0.000 }
gfCNCPoint6[3582] = {X 62.9996, Y 9.4933, Z -8.0000, A 0.000, B 0.000, C 0.000 }
gfCNCPoint6[3583] = {X 63.5143, Y 10.3124, Z -8.0000, A 0.000, B 0.000, C 0.000 }
gfCNCPoint6[3584] = {X 63.8338, Y 11.2255, Z -8.0000, A 0.000, B 0.000, C 0.000 }
gfCNCPoint6[3585] = {X 63.9421, Y 12.1868, Z -8.0000, A 0.000, B 0.000, C 0.000 }
gfCNCPoint6[3586] = {X 63.9421, Y 12.9782, Z -8.0000, A 0.000, B 0.000, C 0.000 }
gfCNCPoint6[3587] = {X 63.8584, Y 13.8244, Z -8.0000, A 0.000, B 0.000, C 0.000 }
gfCNCPoint6[3588] = {X 63.6106, Y 14.6377, Z -8.0000, A 0.000, B 0.000, C 0.000 }
gfCNCPoint6[3589] = {X 63.2082, Y 15.3868, Z -8.0000, A 0.000, B 0.000, C 0.000 }
gfCNCPoint6[3590] = {X 63.4271, Y 15.9632, Z -8.0000, A 0.000, B 0.000, C 0.000 }
gfCNCPoint6[3591] = {X 66.2401, Y 23.4298, Z -8.0000, A 0.000, B 0.000, C 0.000 }
gfCNCPoint6[3592] = {X 72.2110, Y 39.5004, Z -8.0000, A 0.000, B 0.000, C 0.000 }
gfCNCPoint6[3593] = {X 72.5166, Y 40.2690, Z -8.0000, A 0.000, B 0.000, C 0.000 }
gfCNCPoint6[3594] = {X 73.3605, Y 40.7710, Z -8.0000, A 0.000, B 0.000, C 0.000 }
gfCNCPoint6[3595] = {X 74.0693, Y 41.4505, Z -8.0000, A 0.000, B 0.000, C 0.000 }
gfCNCPoint6[3596] = {X 74.6063, Y 42.2726, Z -8.0000, A 0.000, B 0.000, C 0.000 }
gfCNCPoint6[3597] = {X 74.9437, Y 43.1947, Z -8.0000, A 0.000, B 0.000, C 0.000 }
gfCNCPoint6[3598] = {X 75.0643, Y 44.1692, Z -8.0000, A 0.000, B 0.000, C 0.000 }
gfCNCPoint6[3599] = {X 75.0645, Y 45.0000, Z -8.0000, A 0.000, B 0.000, C 0.000 }
gfCNCPoint6[3600] = {X 74.9561, Y 45.9613, Z -8.0000, A 0.000, B 0.000, C 0.000 }
gfCNCPoint6[3601] = {X 74.6366, Y 46.8744, Z -8.0000, A 0.000, B 0.000, C 0.000 }
gfCNCPoint6[3602] = {X 74.1220, Y 47.6935, Z -8.0000, A 0.000, B 0.000, C 0.000 }
gfCNCPoint6[3603] = {X 73.4379, Y 48.3775, Z -8.0000, A 0.000, B 0.000, C 0.000 }
gfCNCPoint6[3604] = {X 72.6188, Y 48.8922, Z -8.0000, A 0.000, B 0.000, C 0.000 }
gfCNCPoint6[3605] = {X 71.7057, Y 49.2117, Z -8.0000, A 0.000, B 0.000, C 0.000 }
gfCNCPoint6[3606] = {X 70.7445, Y 49.3200, Z -8.0000, A 0.000, B 0.000, C 0.000 }
gfCNCPoint6[3607] = {X 64.1851, Y 49.3200, Z -8.0000, A 0.000, B 0.000, C 0.000 }
gfCNCPoint6[3608] = {X 63.2238, Y 49.2117, Z -8.0000, A 0.000, B 0.000, C 0.000 }
gfCNCPoint6[3609] = {X 62.3108, Y 48.8922, Z -8.0000, A 0.000, B 0.000, C 0.000 }
gfCNCPoint6[3610] = {X 61.4917, Y 48.3775, Z -8.0000, A 0.000, B 0.000, C 0.000 }
gfCNCPoint6[3611] = {X 60.8076, Y 47.6935, Z -8.0000, A 0.000, B 0.000, C 0.000 }
gfCNCPoint6[3612] = {X 60.2929, Y 46.8744, Z -8.0000, A 0.000, B 0.000, C 0.000 }
gfCNCPoint6[3613] = {X 59.9734, Y 45.9613, Z -8.0000, A 0.000, B 0.000, C 0.000 }
gfCNCPoint6[3614] = {X 59.8651, Y 45.0000, Z -8.0000, A 0.000, B 0.000, C 0.000 }
gfCNCPoint6[3615] = {X 59.8651, Y 44.2085, Z -8.0000, A 0.000, B 0.000, C 0.000 }
gfCNCPoint6[3616] = {X 59.9515, Y 43.3503, Z -8.0000, A 0.000, B 0.000, C 0.000 }
gfCNCPoint6[3617] = {X 60.2067, Y 42.5264, Z -8.0000, A 0.000, B 0.000, C 0.000 }
gfCNCPoint6[3618] = {X 60.6205, Y 41.7696, Z -8.0000, A 0.000, B 0.000, C 0.000 }
gfCNCPoint6[3619] = {X 60.0064, Y 40.0892, Z -8.0000, A 0.000, B 0.000, C 0.000 }
gfCNCPoint6[3620] = {X 52.0785, Y 40.0892, Z -8.0000, A 0.000, B 0.000, C 0.000 }
gfCNCPoint6[3621] = {X 51.3353, Y 42.0861, Z -8.0000, A 0.000, B 0.000, C 0.000 }
gfCNCPoint6[3622] = {X 51.3382, Y 42.0910, Z -8.0000, A 0.000, B 0.000, C 0.000 }
gfCNCPoint6[3623] = {X 51.6392, Y 42.7502, Z -8.0000, A 0.000, B 0.000, C 0.000 }
gfCNCPoint6[3624] = {X 51.8258, Y 43.4504, Z -8.0000, A 0.000, B 0.000, C 0.000 }
gfCNCPoint6[3625] = {X 51.8928, Y 44.1720, Z -8.0000, A 0.000, B 0.000, C 0.000 }
gfCNCPoint6[3626] = {X 51.8929, Y 45.0000, Z -8.0000, A 0.000, B 0.000, C 0.000 }
gfCNCPoint6[3627] = {X 51.7846, Y 45.9613, Z -8.0000, A 0.000, B 0.000, C 0.000 }
gfCNCPoint6[3628] = {X 51.4651, Y 46.8744, Z -8.0000, A 0.000, B 0.000, C 0.000 }
gfCNCPoint6[3629] = {X 50.9504, Y 47.6935, Z -8.0000, A 0.000, B 0.000, C 0.000 }
gfCNCPoint6[3630] = {X 50.2664, Y 48.3775, Z -8.0000, A 0.000, B 0.000, C 0.000 }
gfCNCPoint6[3631] = {X 49.4473, Y 48.8922, Z -8.0000, A 0.000, B 0.000, C 0.000 }
gfCNCPoint6[3632] = {X 48.5342, Y 49.2117, Z -8.0000, A 0.000, B 0.000, C 0.000 }
gfCNCPoint6[3633] = {X 47.5729, Y 49.3200, Z -8.0000, A 0.000, B 0.000, C 0.000 }
gfCNCPoint6[3634] = {X 40.6393, Y 49.3200, Z -8.0000, A 0.000, B 0.000, C 0.000 }
gfCNCPoint6[3635] = {X 39.6780, Y 49.2117, Z -8.0000, A 0.000, B 0.000, C 0.000 }
gfCNCPoint6[3636] = {X 38.7649, Y 48.8922, Z -8.0000, A 0.000, B 0.000, C 0.000 }
gfCNCPoint6[3637] = {X 37.9458, Y 48.3775, Z -8.0000, A 0.000, B 0.000, C 0.000 }
gfCNCPoint6[3638] = {X 37.2618, Y 47.6935, Z -8.0000, A 0.000, B 0.000, C 0.000 }
gfCNCPoint6[3639] = {X 36.7471, Y 46.8744, Z -8.0000, A 0.000, B 0.000, C 0.000 }
gfCNCPoint6[3640] = {X 36.4276, Y 45.9613, Z -8.0000, A 0.000, B 0.000, C 0.000 }
gfCNCPoint6[3641] = {X 36.3193, Y 45.0000, Z -8.0000, A 0.000, B 0.000, C 0.000 }
gfCNCPoint6[3642] = {X 36.3193, Y 44.2086, Z -8.0000, A 0.000, B 0.000, C 0.000 }
gfCNCPoint6[3643] = {X 36.4359, Y 43.2118, Z -8.0000, A 0.000, B 0.000, C 0.000 }
gfCNCPoint6[3644] = {X 36.7794, Y 42.2688, Z -8.0000, A 0.000, B 0.000, C 0.000 }
gfCNCPoint6[3645] = {X 37.3312, Y 41.4305, Z -8.0000, A 0.000, B 0.000, C 0.000 }
